KUKA KRL program: EPS_2_251806_MH12A_A_20260223023041.src

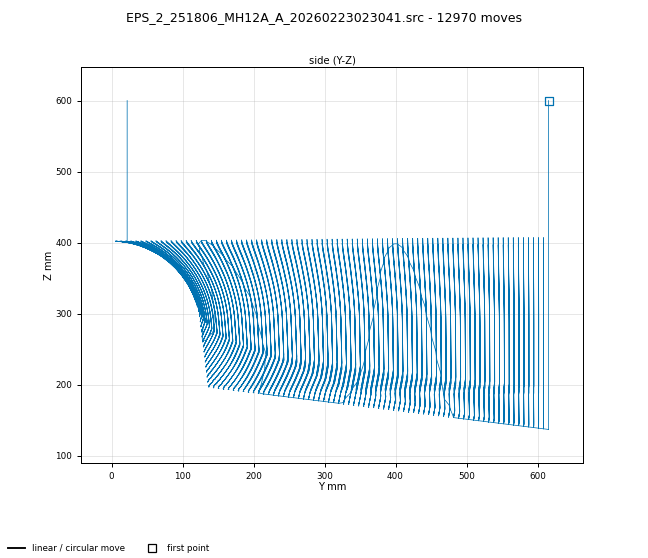
[picture p0: tool path of EPS_2_251806_MH12A_A_20260223023041.src, 12970 of 12972 moves have a stored position in this frame; points joined in program order, loops and branches not executed]
&ACCESS RVP
&REL 4
&COMMENT QRS 19112012
&PARAM EDITMASK = *
DEF PART()
EXT BAS (BAS_COMMAND :IN,REAL :IN )
INT I
BAS (#INITMOV,0 )

;KUKA QRS Post kuka4.cps  Date:22-06-2017 !

File_ID=3069

QRS_PRE_INIT()

;Init var - Until changes are made in qrs_pre_init
Outlet_Square_prg=0
Inlet_1_Square_prg=0
Inlet_2_Square_prg=0
Inlet_3_Square_prg=0
Inlet_4_Square_prg=0
Inlet_5_Square_prg=0

Outlet_1={X 0.000, Y 546.330, Z 306.500, B 0.000, E1 0.000 }
Inlet_1={X 0.000, Y 547.040, Z 296.500, B 0.000, E1 180.000 }
Outlet_1_type=201
Inlet_1_type=201
;QRS#1=Sidecore dimensions
;QRS#2=200-8" PVC SDR 35
;QRS#3=200-8" PVC SDR 35
;QRS#4=
;QRS#5=
;QRS#6=
;QRS#7=
;QRS#8=
;QRS#9=12-08 PSX
;QRS#10=12-08 PSX
;QRS#11=
;QRS#12=
;QRS#13=
;QRS#14=
;QRS#15=
;QRS#16=1220x127x686 2,25'
;QRS#17=EPS Height
;QRS#18=407
;QRS#19=*
;QRS#20= UPDATED VERSION 22-06-2017
;QRS#21=*
Outlet_Square=0100
Inlet_1_Square=0100
Inlet_2_Square=0
Inlet_3_Square=0
Inlet_4_Square=0
Inlet_5_Square=0
Mill_Square=1
Outlet_Square_Prg=204
Inlet_1_Square_prg=204

QRS_INIT()

$ADVANCE=5

; T1
PTP {E1 173.588,E2 173.588}
PTP {X 0,Y 615.517,A -85,B 0,C 180,E1 173.588,E2 173.588,E3 0,E4 0,E5 0,E6 0}
QRS_SPEED_INIT()
LIN {X 0,Y 615.517,Z 600,A -85,B 0,C 180,E1 173.588,E2 173.588,E3 0,E4 0,E5 0,E6 0} C_VEL
LIN {X 0,Y 615.517,Z 146.874,A -85,B 0,C 180,E1 173.588,E2 173.588} C_VEL
LIN {X 0,Y 615.517,Z 138.695,A -85,B 0,C 180,E1 173.588,E2 173.588} C_VEL
LIN {X 0,Y 615.495,Z 136.695,A -85,B 0,C 180,E1 173.402,E2 173.402} C_VEL
LIN {X 0,Y 615.467,Z 136.688,A -85,B 0,C 180,E1 170.801,E2 170.801} C_VEL
LIN {X 0,Y 615.466,Z 136.688,A -85,B 0,C 180,E1 168.806,E2 168.806} C_VEL
LIN {X 0,Y 615.457,Z 136.695,A -85,B 0,C 180,E1 166.125,E2 166.125} C_VEL
LIN {X 0,Y 615.494,Z 136.691,A -85,B 0,C 180,E1 163.413,E2 163.413} C_VEL
LIN {X 0,Y 615.453,Z 136.69,A -85,B 0,C 180,E1 160.661,E2 160.661} C_VEL
LIN {X 0,Y 615.451,Z 136.691,A -85,B 0,C 180,E1 158.567,E2 158.567} C_VEL
LIN {X 0,Y 615.477,Z 136.698,A -85,B 0,C 180,E1 155.99,E2 155.99} C_VEL
LIN {X 0,Y 615.465,Z 136.688,A -85,B 0,C 180,E1 152.956,E2 152.956} C_VEL
LIN {X 0,Y 615.449,Z 136.693,A -85,B 0,C 180,E1 150.592,E2 150.592} C_VEL
LIN {X 0,Y 615.494,Z 136.693,A -85,B 0,C 180,E1 147.666,E2 147.666} C_VEL
LIN {X 0,Y 615.473,Z 136.687,A -85,B 0,C 180,E1 145.184,E2 145.184} C_VEL
LIN {X 0,Y 615.452,Z 136.691,A -85,B 0,C 180,E1 142.755,E2 142.755} C_VEL
LIN {X 0,Y 615.496,Z 136.698,A -85,B 0,C 180,E1 139.908,E2 139.908} C_VEL
LIN {X 0,Y 615.494,Z 136.689,A -85,B 0,C 180,E1 137.647,E2 137.647} C_VEL
LIN {X 0,Y 615.455,Z 136.69,A -85,B 0,C 180,E1 134.928,E2 134.928} C_VEL
LIN {X 0,Y 615.496,Z 136.701,A -85,B 0,C 180,E1 132.081,E2 132.081} C_VEL
LIN {X 0,Y 615.494,Z 136.689,A -85,B 0,C 180,E1 129.748,E2 129.748} C_VEL
LIN {X 0,Y 615.466,Z 136.687,A -85,B 0,C 180,E1 127.242,E2 127.242} C_VEL
LIN {X 0,Y 615.458,Z 136.694,A -85,B 0,C 180,E1 124.696,E2 124.696} C_VEL
LIN {X 0,Y 615.487,Z 136.699,A -85,B 0,C 180,E1 122.33,E2 122.33} C_VEL
LIN {X 0,Y 615.472,Z 136.686,A -85,B 0,C 180,E1 119.406,E2 119.406} C_VEL
LIN {X 0,Y 615.455,Z 136.691,A -85,B 0,C 180,E1 117.038,E2 117.038} C_VEL
LIN {X 0,Y 615.454,Z 136.692,A -85,B 0,C 180,E1 114.992,E2 114.992} C_VEL
LIN {X 0,Y 615.491,Z 136.694,A -85,B 0,C 180,E1 112.135,E2 112.135} C_VEL
LIN {X 0,Y 615.491,Z 136.885,A -85,B 0,C 180,E1 110.293,E2 110.293} C_VEL
LIN {X 0,Y 615.493,Z 154.026,A -85,B 0,C 180,E1 107.612,E2 107.612} C_VEL
LIN {X 0,Y 615.449,Z 171.874,A -85,B 0,C 180,E1 104.888,E2 104.888} C_VEL
LIN {X 0,Y 615.436,Z 185.406,A -85,B 0,C 180,E1 102.866,E2 102.866} C_VEL
LIN {X 0,Y 615.435,Z 186.907,A -85,B 0,C 180,E1 102.803,E2 102.803} C_VEL
LIN {X 0,Y 615.497,Z 292.675,A -85,B 0,C 180,E1 101.547,E2 101.547} C_VEL
LIN {X 0,Y 615.498,Z 305.242,A -85,B 0,C 180,E1 101.276,E2 101.276} C_VEL
LIN {X 0,Y 615.497,Z 318.527,A -85,B 0,C 180,E1 100.845,E2 100.845} C_VEL
LIN {X 0,Y 615.491,Z 329.577,A -85,B 0,C 180,E1 100.36,E2 100.36} C_VEL
LIN {X 0,Y 615.492,Z 341.312,A -85,B 0,C 180,E1 99.696,E2 99.696} C_VEL
LIN {X 0,Y 615.499,Z 351.774,A -85,B 0,C 180,E1 98.95,E2 98.95} C_VEL
LIN {X 0,Y 615.498,Z 360.336,A -85,B 0,C 180,E1 98.205,E2 98.205} C_VEL
LIN {X 0,Y 615.497,Z 368.213,A -85,B 0,C 180,E1 97.38,E2 97.38} C_VEL
LIN {X 0,Y 615.497,Z 375.902,A -85,B 0,C 180,E1 96.392,E2 96.392} C_VEL
LIN {X 0,Y 615.497,Z 382.96,A -85,B 0,C 180,E1 95.241,E2 95.241} C_VEL
LIN {X 0,Y 615.494,Z 387.659,A -85,B 0,C 180,E1 94.256,E2 94.256} C_VEL
LIN {X 0,Y 615.494,Z 391.256,A -85,B 0,C 180,E1 93.273,E2 93.273} C_VEL
LIN {X 0,Y 615.496,Z 393.116,A -85,B 0,C 180,E1 92.617,E2 92.617} C_VEL
LIN {X 0,Y 615.499,Z 394.533,A -85,B 0,C 180,E1 91.963,E2 91.963} C_VEL
LIN {X 0,Y 615.496,Z 396.142,A -85,B 0,C 180,E1 90.654,E2 90.654} C_VEL
LIN {X 0,Y 615.495,Z 396.384,A -85,B 0,C 180,E1 90,E2 90} C_VEL
LIN {X 0,Y 615.495,Z 396.205,A -85,B 0,C 180,E1 89.345,E2 89.345} C_VEL
LIN {X 0,Y 615.499,Z 394.682,A -85,B 0,C 180,E1 88.037,E2 88.037} C_VEL
LIN {X 0,Y 615.498,Z 393.341,A -85,B 0,C 180,E1 87.382,E2 87.382} C_VEL
LIN {X 0,Y 615.496,Z 390.493,A -85,B 0,C 180,E1 86.399,E2 86.399} C_VEL
LIN {X 0,Y 615.498,Z 386.633,A -85,B 0,C 180,E1 85.415,E2 85.415} C_VEL
LIN {X 0,Y 615.498,Z 381.651,A -85,B 0,C 180,E1 84.43,E2 84.43} C_VEL
LIN {X 0,Y 615.496,Z 375.208,A -85,B 0,C 180,E1 83.418,E2 83.418} C_VEL
LIN {X 0,Y 615.497,Z 367.536,A -85,B 0,C 180,E1 82.454,E2 82.454} C_VEL
LIN {X 0,Y 615.498,Z 357.758,A -85,B 0,C 180,E1 81.463,E2 81.463} C_VEL
LIN {X 0,Y 615.498,Z 347.492,A -85,B 0,C 180,E1 80.636,E2 80.636} C_VEL
LIN {X 0,Y 615.486,Z 335.93,A -85,B 0,C 180,E1 79.889,E2 79.889} C_VEL
LIN {X 0,Y 615.497,Z 324.023,A -85,B 0,C 180,E1 79.291,E2 79.291} C_VEL
LIN {X 0,Y 615.498,Z 311.157,A -85,B 0,C 180,E1 78.807,E2 78.807} C_VEL
LIN {X 0,Y 615.497,Z 298.557,A -85,B 0,C 180,E1 78.473,E2 78.473} C_VEL
LIN {X 0,Y 615.495,Z 285.433,A -85,B 0,C 180,E1 78.265,E2 78.265} C_VEL
LIN {X 0,Y 615.429,Z 186.202,A -85,B 0,C 180,E1 77.091,E2 77.091} C_VEL
LIN {X 0,Y 615.434,Z 184.751,A -85,B 0,C 180,E1 76.966,E2 76.966} C_VEL
LIN {X 0,Y 615.496,Z 166.877,A -85,B 0,C 180,E1 74.265,E2 74.265} C_VEL
LIN {X 0,Y 615.455,Z 149.286,A -85,B 0,C 180,E1 71.565,E2 71.565} C_VEL
LIN {X 0,Y 615.497,Z 136.85,A -85,B 0,C 180,E1 69.608,E2 69.608} C_VEL
LIN {X 0,Y 615.464,Z 136.695,A -85,B 0,C 180,E1 67.155,E2 67.155} C_VEL
LIN {X 0,Y 615.483,Z 136.684,A -85,B 0,C 180,E1 64.433,E2 64.433} C_VEL
LIN {X 0,Y 615.489,Z 136.699,A -85,B 0,C 180,E1 61.55,E2 61.55} C_VEL
LIN {X 0,Y 615.46,Z 136.69,A -85,B 0,C 180,E1 58.919,E2 58.919} C_VEL
LIN {X 0,Y 615.488,Z 136.683,A -85,B 0,C 180,E1 56.466,E2 56.466} C_VEL
LIN {X 0,Y 615.481,Z 136.698,A -85,B 0,C 180,E1 53.575,E2 53.575} C_VEL
LIN {X 0,Y 615.458,Z 136.689,A -85,B 0,C 180,E1 50.942,E2 50.942} C_VEL
LIN {X 0,Y 615.489,Z 136.684,A -85,B 0,C 180,E1 48.527,E2 48.527} C_VEL
LIN {X 0,Y 615.497,Z 136.701,A -85,B 0,C 180,E1 45.852,E2 45.852} C_VEL
LIN {X 0,Y 615.46,Z 136.689,A -85,B 0,C 180,E1 43.046,E2 43.046} C_VEL
LIN {X 0,Y 615.489,Z 136.684,A -85,B 0,C 180,E1 40.607,E2 40.607} C_VEL
LIN {X 0,Y 615.484,Z 136.702,A -85,B 0,C 180,E1 38.013,E2 38.013} C_VEL
LIN {X 0,Y 615.465,Z 136.696,A -85,B 0,C 180,E1 35.618,E2 35.618} C_VEL
LIN {X 0,Y 615.456,Z 136.69,A -85,B 0,C 180,E1 33.238,E2 33.238} C_VEL
LIN {X 0,Y 615.473,Z 136.686,A -85,B 0,C 180,E1 30.921,E2 30.921} C_VEL
LIN {X 0,Y 615.48,Z 136.698,A -85,B 0,C 180,E1 27.916,E2 27.916} C_VEL
LIN {X 0,Y 615.456,Z 136.693,A -85,B 0,C 180,E1 25.565,E2 25.565} C_VEL
LIN {X 0,Y 615.488,Z 136.684,A -85,B 0,C 180,E1 22.845,E2 22.845} C_VEL
LIN {X 0,Y 615.481,Z 136.698,A -85,B 0,C 180,E1 20.033,E2 20.033} C_VEL
LIN {X 0,Y 615.469,Z 136.697,A -85,B 0,C 180,E1 17.958,E2 17.958} C_VEL
LIN {X 0,Y 615.464,Z 136.696,A -85,B 0,C 180,E1 15.906,E2 15.906} C_VEL
LIN {X 0,Y 615.466,Z 136.687,A -85,B 0,C 180,E1 13.202,E2 13.202} C_VEL
LIN {X 0,Y 615.494,Z 136.694,A -85,B 0,C 180,E1 10.527,E2 10.527} C_VEL
LIN {X 0,Y 615.457,Z 136.695,A -85,B 0,C 180,E1 7.876,E2 7.876} C_VEL
LIN {X 0,Y 615.469,Z 136.687,A -85,B 0,C 180,E1 5.241,E2 5.241} C_VEL
LIN {X 0,Y 615.494,Z 136.695,A -85,B 0,C 180,E1 2.618,E2 2.618} C_VEL
LIN {X 0,Y 615.457,Z 136.695,A -85,B 0,C 180,E1 0,E2 0} C_VEL
LIN {X 0,Y 615.464,Z 136.688,A -85,B 0,C 180,E1 -2.618,E2 -2.618} C_VEL
LIN {X 0,Y 615.494,Z 136.693,A -85,B 0,C 180,E1 -5.241,E2 -5.241} C_VEL
LIN {X 0,Y 615.456,Z 136.696,A -85,B 0,C 180,E1 -7.876,E2 -7.876} C_VEL
LIN {X 0,Y 615.463,Z 136.688,A -85,B 0,C 180,E1 -10.527,E2 -10.527} C_VEL
LIN {X 0,Y 615.495,Z 136.695,A -85,B 0,C 180,E1 -13.201,E2 -13.201} C_VEL
LIN {X 0,Y 615.451,Z 136.694,A -85,B 0,C 180,E1 -15.906,E2 -15.906} C_VEL
LIN {X 0,Y 615.448,Z 136.694,A -85,B 0,C 180,E1 -17.958,E2 -17.958} C_VEL
LIN {X 0,Y 615.49,Z 136.687,A -85,B 0,C 180,E1 -20.731,E2 -20.731} C_VEL
LIN {X 0,Y 615.464,Z 136.697,A -85,B 0,C 180,E1 -23.557,E2 -23.557} C_VEL
LIN {X 0,Y 615.451,Z 136.695,A -85,B 0,C 180,E1 -25.717,E2 -25.717} C_VEL
LIN {X 0,Y 615.447,Z 136.693,A -85,B 0,C 180,E1 -27.917,E2 -27.917} C_VEL
LIN {X 0,Y 615.449,Z 136.691,A -85,B 0,C 180,E1 -30.162,E2 -30.162} C_VEL
LIN {X 0,Y 615.478,Z 136.687,A -85,B 0,C 180,E1 -32.458,E2 -32.458} C_VEL
LIN {X 0,Y 615.495,Z 136.692,A -85,B 0,C 180,E1 -34.815,E2 -34.815} C_VEL
LIN {X 0,Y 615.474,Z 136.698,A -85,B 0,C 180,E1 -37.243,E2 -37.243} C_VEL
LIN {X 0,Y 615.445,Z 136.693,A -85,B 0,C 180,E1 -39.754,E2 -39.754} C_VEL
LIN {X 0,Y 615.478,Z 136.688,A -85,B 0,C 180,E1 -42.354,E2 -42.354} C_VEL
LIN {X 0,Y 615.482,Z 136.699,A -85,B 0,C 180,E1 -45.069,E2 -45.069} C_VEL
LIN {X 0,Y 615.444,Z 136.694,A -85,B 0,C 180,E1 -47.644,E2 -47.644} C_VEL
LIN {X 0,Y 615.476,Z 136.688,A -85,B 0,C 180,E1 -50.25,E2 -50.25} C_VEL
LIN {X 0,Y 615.47,Z 136.698,A -85,B 0,C 180,E1 -53.066,E2 -53.066} C_VEL
LIN {X 0,Y 615.45,Z 136.696,A -85,B 0,C 180,E1 -55.305,E2 -55.305} C_VEL
LIN {X 0,Y 615.443,Z 136.693,A -85,B 0,C 180,E1 -57.676,E2 -57.676} C_VEL
LIN {X 0,Y 615.482,Z 136.688,A -85,B 0,C 180,E1 -60.207,E2 -60.207} C_VEL
LIN {X 0,Y 615.467,Z 136.698,A -85,B 0,C 180,E1 -62.959,E2 -62.959} C_VEL
LIN {X 0,Y 615.46,Z 136.697,A -85,B 0,C 180,E1 -65.007,E2 -65.007} C_VEL
LIN {X 0,Y 615.446,Z 136.696,A -85,B 0,C 180,E1 -67.154,E2 -67.154} C_VEL
LIN {X 0,Y 615.494,Z 136.913,A -85,B 0,C 180,E1 -68.7,E2 -68.7} C_VEL
LIN {X 0,Y 615.486,Z 153.668,A -85,B 0,C 180,E1 -71.181,E2 -71.181} C_VEL
LIN {X 0,Y 615.486,Z 173.832,A -85,B 0,C 180,E1 -74.095,E2 -74.095} C_VEL
LIN {X 0,Y 615.479,Z 193.975,A -85,B 0,C 180,E1 -76.967,E2 -76.967} C_VEL
LIN {X 0,Y 615.486,Z 195.337,A -85,B 0,C 180,E1 -77.114,E2 -77.114} C_VEL
LIN {X 0,Y 615.487,Z 202.259,A -85,B 0,C 180,E1 -77.218,E2 -77.218} C_VEL
LIN {X 0,Y 615.498,Z 302.827,A -85,B 0,C 180,E1 -78.411,E2 -78.411} C_VEL
LIN {X 0,Y 615.498,Z 315.341,A -85,B 0,C 180,E1 -78.682,E2 -78.682} C_VEL
LIN {X 0,Y 615.496,Z 328.502,A -85,B 0,C 180,E1 -79.109,E2 -79.109} C_VEL
LIN {X 0,Y 615.489,Z 340.476,A -85,B 0,C 180,E1 -79.639,E2 -79.639} C_VEL
LIN {X 0,Y 615.495,Z 351.993,A -85,B 0,C 180,E1 -80.304,E2 -80.304} C_VEL
LIN {X 0,Y 615.499,Z 362.34,A -85,B 0,C 180,E1 -81.05,E2 -81.05} C_VEL
LIN {X 0,Y 615.497,Z 370.811,A -85,B 0,C 180,E1 -81.794,E2 -81.794} C_VEL
LIN {X 0,Y 615.498,Z 378.605,A -85,B 0,C 180,E1 -82.619,E2 -82.619} C_VEL
LIN {X 0,Y 615.496,Z 386.202,A -85,B 0,C 180,E1 -83.608,E2 -83.608} C_VEL
LIN {X 0,Y 615.498,Z 393.204,A -85,B 0,C 180,E1 -84.759,E2 -84.759} C_VEL
LIN {X 0,Y 615.494,Z 397.85,A -85,B 0,C 180,E1 -85.743,E2 -85.743} C_VEL
LIN {X 0,Y 615.494,Z 401.398,A -85,B 0,C 180,E1 -86.727,E2 -86.727} C_VEL
LIN {X 0,Y 615.497,Z 403.232,A -85,B 0,C 180,E1 -87.382,E2 -87.382} C_VEL
LIN {X 0,Y 615.499,Z 404.607,A -85,B 0,C 180,E1 -88.037,E2 -88.037} C_VEL
LIN {X 0,Y 615.496,Z 406.173,A -85,B 0,C 180,E1 -89.345,E2 -89.345} C_VEL
LIN {X 0,Y 615.494,Z 406.389,A -85,B 0,C 180,E1 -90,E2 -90} C_VEL
LIN {X 0,Y 615.495,Z 405.58,A -85,B 0,C 180,E1 -91.308,E2 -91.308} C_VEL
LIN {X 0,Y 615.499,Z 404.608,A -85,B 0,C 180,E1 -91.963,E2 -91.963} C_VEL
LIN {X 0,Y 615.497,Z 403.234,A -85,B 0,C 180,E1 -92.617,E2 -92.617} C_VEL
LIN {X 0,Y 615.496,Z 400.351,A -85,B 0,C 180,E1 -93.6,E2 -93.6} C_VEL
LIN {X 0,Y 615.498,Z 396.443,A -85,B 0,C 180,E1 -94.584,E2 -94.584} C_VEL
LIN {X 0,Y 615.499,Z 391.407,A -85,B 0,C 180,E1 -95.569,E2 -95.569} C_VEL
LIN {X 0,Y 615.496,Z 384.87,A -85,B 0,C 180,E1 -96.583,E2 -96.583} C_VEL
LIN {X 0,Y 615.497,Z 377.137,A -85,B 0,C 180,E1 -97.545,E2 -97.545} C_VEL
LIN {X 0,Y 615.498,Z 369.05,A -85,B 0,C 180,E1 -98.371,E2 -98.371} C_VEL
LIN {X 0,Y 615.499,Z 359.174,A -85,B 0,C 180,E1 -99.198,E2 -99.198} C_VEL
LIN {X 0,Y 615.492,Z 347.989,A -85,B 0,C 180,E1 -99.945,E2 -99.945} C_VEL
LIN {X 0,Y 615.493,Z 337.033,A -85,B 0,C 180,E1 -100.526,E2 -100.526} C_VEL
LIN {X 0,Y 615.499,Z 324.425,A -85,B 0,C 180,E1 -101.042,E2 -101.042} C_VEL
LIN {X 0,Y 615.499,Z 312.087,A -85,B 0,C 180,E1 -101.401,E2 -101.401} C_VEL
LIN {X 0,Y 615.499,Z 298.504,A -85,B 0,C 180,E1 -101.651,E2 -101.651} C_VEL
LIN {X 0,Y 615.486,Z 195.821,A -85,B 0,C 180,E1 -102.865,E2 -102.865} C_VEL
LIN {X 0,Y 615.484,Z 194.624,A -85,B 0,C 180,E1 -102.949,E2 -102.949} C_VEL
LIN {X 0,Y 615.491,Z 175.021,A -85,B 0,C 180,E1 -105.734,E2 -105.734} C_VEL
LIN {X 0,Y 615.476,Z 155.169,A -85,B 0,C 180,E1 -108.601,E2 -108.601} C_VEL
LIN {X 0,Y 615.494,Z 137.129,A -85,B 0,C 180,E1 -111.255,E2 -111.255} C_VEL
LIN {X 0,Y 615.498,Z 136.727,A -85,B 0,C 180,E1 -111.431,E2 -111.431} C_VEL
LIN {X 0,Y 615.446,Z 136.692,A -85,B 0,C 180,E1 -114.273,E2 -114.273} C_VEL
LIN {X 0,Y 615.441,Z 136.693,A -85,B 0,C 180,E1 -116.445,E2 -116.445} C_VEL
LIN {X 0,Y 615.444,Z 136.695,A -85,B 0,C 180,E1 -118.659,E2 -118.659} C_VEL
LIN {X 0,Y 615.476,Z 136.699,A -85,B 0,C 180,E1 -121.084,E2 -121.084} C_VEL
LIN {X 0,Y 615.456,Z 136.69,A -85,B 0,C 180,E1 -124.023,E2 -124.023} C_VEL
LIN {X 0,Y 615.442,Z 136.694,A -85,B 0,C 180,E1 -126.427,E2 -126.427} C_VEL
LIN {X 0,Y 615.487,Z 136.699,A -85,B 0,C 180,E1 -129.062,E2 -129.062} C_VEL
LIN {X 0,Y 615.495,Z 136.69,A -85,B 0,C 180,E1 -131.472,E2 -131.472} C_VEL
LIN {X 0,Y 615.445,Z 136.692,A -85,B 0,C 180,E1 -134.152,E2 -134.152} C_VEL
LIN {X 0,Y 615.485,Z 136.699,A -85,B 0,C 180,E1 -136.951,E2 -136.951} C_VEL
LIN {X 0,Y 615.494,Z 136.689,A -85,B 0,C 180,E1 -139.394,E2 -139.394} C_VEL
LIN {X 0,Y 615.448,Z 136.691,A -85,B 0,C 180,E1 -141.991,E2 -141.991} C_VEL
LIN {X 0,Y 615.448,Z 136.695,A -85,B 0,C 180,E1 -144.381,E2 -144.381} C_VEL
LIN {X 0,Y 615.47,Z 136.7,A -85,B 0,C 180,E1 -146.763,E2 -146.763} C_VEL
LIN {X 0,Y 615.492,Z 136.695,A -85,B 0,C 180,E1 -149.08,E2 -149.08} C_VEL
LIN {X 0,Y 615.471,Z 136.688,A -85,B 0,C 180,E1 -151.549,E2 -151.549} C_VEL
LIN {X 0,Y 615.466,Z 136.689,A -85,B 0,C 180,E1 -153.555,E2 -153.555} C_VEL
LIN {X 0,Y 615.445,Z 136.692,A -85,B 0,C 180,E1 -155.997,E2 -155.997} C_VEL
LIN {X 0,Y 615.473,Z 136.698,A -85,B 0,C 180,E1 -158.568,E2 -158.568} C_VEL
LIN {X 0,Y 615.475,Z 136.688,A -85,B 0,C 180,E1 -161.394,E2 -161.394} C_VEL
LIN {X 0,Y 615.459,Z 136.689,A -85,B 0,C 180,E1 -163.572,E2 -163.572} C_VEL
LIN {X 0,Y 615.45,Z 136.695,A -85,B 0,C 180,E1 -166.125,E2 -166.125} C_VEL
LIN {X 0,Y 615.493,Z 136.696,A -85,B 0,C 180,E1 -168.807,E2 -168.807} C_VEL
LIN {X 0,Y 615.457,Z 136.69,A -85,B 0,C 180,E1 -171.463,E2 -171.463} C_VEL
LIN {X 0,Y 615.461,Z 136.689,A -85,B 0,C 180,E1 -173.443,E2 -173.443} C_VEL
LIN {X 0,Y 615.454,Z 136.695,A -85,B 0,C 180,E1 -176.071,E2 -176.071} C_VEL
LIN {X 0,Y 615.495,Z 136.695,A -85,B 0,C 180,E1 -178.691,E2 -178.691} C_VEL
LIN {X 0,Y 615.465,Z 136.688,A -85,B 0,C 180,E1 -181.309,E2 -181.309} C_VEL
LIN {X 0,Y 615.453,Z 136.695,A -85,B 0,C 180,E1 -183.929,E2 -183.929} C_VEL
LIN {X 0,Y 615.495,Z 136.695,A -85,B 0,C 180,E1 -186.598,E2 -186.598} C_VEL
LIN {X 0,Y 614.801,Z 136.835,A -85,B 0,C 180,E1 -187.144,E2 -187.144} C_VEL
LIN {X 0,Y 611.954,Z 137.255,A -85,B 0,C 180,E1 -188.03,E2 -188.03} C_VEL
LIN {X 0,Y 609.562,Z 137.562,A -85,B 0,C 180,E1 -188.742,E2 -188.742} C_VEL
LIN {X 0,Y 608.526,Z 137.679,A -85,B 0,C 180,E1 -189.292,E2 -189.292} C_VEL
LIN {X 0,Y 608.437,Z 137.689,A -85,B 0,C 180,E1 -189.478,E2 -189.478} C_VEL
LIN {X 0,Y 608.44,Z 137.693,A -85,B 0,C 180,E1 -192,E2 -192} C_VEL
LIN {X 0,Y 608.472,Z 137.689,A -85,B 0,C 180,E1 -194.721,E2 -194.721} C_VEL
LIN {X 0,Y 608.427,Z 137.691,A -85,B 0,C 180,E1 -197.477,E2 -197.477} C_VEL
LIN {X 0,Y 608.428,Z 137.691,A -85,B 0,C 180,E1 -199.572,E2 -199.572} C_VEL
LIN {X 0,Y 608.447,Z 137.69,A -85,B 0,C 180,E1 -201.692,E2 -201.692} C_VEL
LIN {X 0,Y 608.448,Z 137.692,A -85,B 0,C 180,E1 -204.571,E2 -204.571} C_VEL
LIN {X 0,Y 608.43,Z 137.691,A -85,B 0,C 180,E1 -207.519,E2 -207.519} C_VEL
LIN {X 0,Y 608.476,Z 137.692,A -85,B 0,C 180,E1 -209.976,E2 -209.976} C_VEL
LIN {X 0,Y 608.443,Z 137.689,A -85,B 0,C 180,E1 -212.881,E2 -212.881} C_VEL
LIN {X 0,Y 608.422,Z 137.691,A -85,B 0,C 180,E1 -215.279,E2 -215.279} C_VEL
LIN {X 0,Y 608.465,Z 137.693,A -85,B 0,C 180,E1 -218.242,E2 -218.242} C_VEL
LIN {X 0,Y 608.474,Z 137.69,A -85,B 0,C 180,E1 -220.334,E2 -220.334} C_VEL
LIN {X 0,Y 608.428,Z 137.69,A -85,B 0,C 180,E1 -222.962,E2 -222.962} C_VEL
LIN {X 0,Y 608.455,Z 137.694,A -85,B 0,C 180,E1 -225.737,E2 -225.737} C_VEL
LIN {X 0,Y 608.452,Z 137.688,A -85,B 0,C 180,E1 -228.659,E2 -228.659} C_VEL
LIN {X 0,Y 608.466,Z 137.695,A -85,B 0,C 180,E1 -231.76,E2 -231.76} C_VEL
LIN {X 0,Y 608.437,Z 137.689,A -85,B 0,C 180,E1 -234.723,E2 -234.723} C_VEL
LIN {X 0,Y 608.442,Z 137.69,A -85,B 0,C 180,E1 -237.121,E2 -237.121} C_VEL
LIN {X 0,Y 608.474,Z 137.69,A -85,B 0,C 180,E1 -240.028,E2 -240.028} C_VEL
LIN {X 0,Y 608.456,Z 137.687,A -85,B 0,C 180,E1 -242.797,E2 -242.797} C_VEL
LIN {X 0,Y 608.444,Z 137.695,A -85,B 0,C 180,E1 -245.429,E2 -245.429} C_VEL
LIN {X 0,Y 608.459,Z 137.688,A -85,B 0,C 180,E1 -248.309,E2 -248.309} C_VEL
LIN {X 0,Y 608.495,Z 137.899,A -85,B 0,C 180,E1 -249.629,E2 -249.629} C_VEL
LIN {X 0,Y 608.506,Z 154.095,A -85,B 0,C 180,E1 -252.179,E2 -252.179} C_VEL
LIN {X 0,Y 608.448,Z 171.991,A -85,B 0,C 180,E1 -254.937,E2 -254.937} C_VEL
LIN {X 0,Y 608.455,Z 185.735,A -85,B 0,C 180,E1 -257.005,E2 -257.005} C_VEL
LIN {X 0,Y 608.528,Z 188.555,A -85,B 0,C 180,E1 -257.07,E2 -257.07} C_VEL
LIN {X 0,Y 608.557,Z 292.826,A -85,B 0,C 180,E1 -258.32,E2 -258.32} C_VEL
LIN {X 0,Y 608.538,Z 306.134,A -85,B 0,C 180,E1 -258.615,E2 -258.615} C_VEL
LIN {X 0,Y 608.529,Z 319.355,A -85,B 0,C 180,E1 -259.055,E2 -259.055} C_VEL
LIN {X 0,Y 608.503,Z 331.379,A -85,B 0,C 180,E1 -259.604,E2 -259.604} C_VEL
LIN {X 0,Y 608.506,Z 342.798,A -85,B 0,C 180,E1 -260.276,E2 -260.276} C_VEL
LIN {X 0,Y 608.474,Z 353.09,A -85,B 0,C 180,E1 -261.03,E2 -261.03} C_VEL
LIN {X 0,Y 608.464,Z 362.354,A -85,B 0,C 180,E1 -261.866,E2 -261.866} C_VEL
LIN {X 0,Y 608.466,Z 371.327,A -85,B 0,C 180,E1 -262.868,E2 -262.868} C_VEL
LIN {X 0,Y 608.444,Z 378.558,A -85,B 0,C 180,E1 -263.867,E2 -263.867} C_VEL
LIN {X 0,Y 608.462,Z 383.437,A -85,B 0,C 180,E1 -264.699,E2 -264.699} C_VEL
LIN {X 0,Y 608.439,Z 388.18,A -85,B 0,C 180,E1 -265.695,E2 -265.695} C_VEL
LIN {X 0,Y 608.425,Z 391.813,A -85,B 0,C 180,E1 -266.689,E2 -266.689} C_VEL
LIN {X 0,Y 608.425,Z 393.692,A -85,B 0,C 180,E1 -267.352,E2 -267.352} C_VEL
LIN {X 0,Y 608.444,Z 395.127,A -85,B 0,C 180,E1 -268.015,E2 -268.015} C_VEL
LIN {X 0,Y 608.439,Z 396.752,A -85,B 0,C 180,E1 -269.338,E2 -269.338} C_VEL
LIN {X 0,Y 608.435,Z 396.995,A -85,B 0,C 180,E1 -270,E2 -270} C_VEL
LIN {X 0,Y 608.438,Z 396.815,A -85,B 0,C 180,E1 -270.662,E2 -270.662} C_VEL
LIN {X 0,Y 608.444,Z 395.276,A -85,B 0,C 180,E1 -271.986,E2 -271.986} C_VEL
LIN {X 0,Y 608.426,Z 393.918,A -85,B 0,C 180,E1 -272.648,E2 -272.648} C_VEL
LIN {X 0,Y 608.449,Z 391.041,A -85,B 0,C 180,E1 -273.643,E2 -273.643} C_VEL
LIN {X 0,Y 608.433,Z 387.142,A -85,B 0,C 180,E1 -274.638,E2 -274.638} C_VEL
LIN {X 0,Y 608.45,Z 382.111,A -85,B 0,C 180,E1 -275.635,E2 -275.635} C_VEL
LIN {X 0,Y 608.441,Z 375.794,A -85,B 0,C 180,E1 -276.633,E2 -276.633} C_VEL
LIN {X 0,Y 608.475,Z 367.877,A -85,B 0,C 180,E1 -277.633,E2 -277.633} C_VEL
LIN {X 0,Y 608.472,Z 358.035,A -85,B 0,C 180,E1 -278.636,E2 -278.636} C_VEL
LIN {X 0,Y 608.48,Z 347.713,A -85,B 0,C 180,E1 -279.473,E2 -279.473} C_VEL
LIN {X 0,Y 608.483,Z 336.099,A -85,B 0,C 180,E1 -280.229,E2 -280.229} C_VEL
LIN {X 0,Y 608.529,Z 324.86,A -85,B 0,C 180,E1 -280.803,E2 -280.803} C_VEL
LIN {X 0,Y 608.538,Z 312.26,A -85,B 0,C 180,E1 -281.29,E2 -281.29} C_VEL
LIN {X 0,Y 608.539,Z 299.559,A -85,B 0,C 180,E1 -281.639,E2 -281.639} C_VEL
LIN {X 0,Y 608.564,Z 287.289,A -85,B 0,C 180,E1 -281.85,E2 -281.85} C_VEL
LIN {X 0,Y 608.484,Z 186.214,A -85,B 0,C 180,E1 -283.059,E2 -283.059} C_VEL
LIN {X 0,Y 608.425,Z 184.884,A -85,B 0,C 180,E1 -283.187,E2 -283.187} C_VEL
LIN {X 0,Y 608.487,Z 166.979,A -85,B 0,C 180,E1 -285.921,E2 -285.921} C_VEL
LIN {X 0,Y 608.466,Z 150.674,A -85,B 0,C 180,E1 -288.445,E2 -288.445} C_VEL
LIN {X 0,Y 608.505,Z 137.841,A -85,B 0,C 180,E1 -290.471,E2 -290.471} C_VEL
LIN {X 0,Y 608.438,Z 137.69,A -85,B 0,C 180,E1 -293.124,E2 -293.124} C_VEL
LIN {X 0,Y 608.477,Z 137.686,A -85,B 0,C 180,E1 -295.721,E2 -295.721} C_VEL
LIN {X 0,Y 608.468,Z 137.691,A -85,B 0,C 180,E1 -298.619,E2 -298.619} C_VEL
LIN {X 0,Y 608.442,Z 137.688,A -85,B 0,C 180,E1 -301.317,E2 -301.317} C_VEL
LIN {X 0,Y 608.475,Z 137.687,A -85,B 0,C 180,E1 -303.735,E2 -303.735} C_VEL
LIN {X 0,Y 608.477,Z 137.692,A -85,B 0,C 180,E1 -306.09,E2 -306.09} C_VEL
LIN {X 0,Y 608.427,Z 137.695,A -85,B 0,C 180,E1 -308.59,E2 -308.59} C_VEL
LIN {X 0,Y 608.454,Z 137.687,A -85,B 0,C 180,E1 -311.341,E2 -311.341} C_VEL
LIN {X 0,Y 608.461,Z 137.695,A -85,B 0,C 180,E1 -314.264,E2 -314.264} C_VEL
LIN {X 0,Y 608.431,Z 137.69,A -85,B 0,C 180,E1 -317.038,E2 -317.038} C_VEL
LIN {X 0,Y 608.457,Z 137.691,A -85,B 0,C 180,E1 -319.697,E2 -319.697} C_VEL
LIN {X 0,Y 608.46,Z 137.693,A -85,B 0,C 180,E1 -322.253,E2 -322.253} C_VEL
LIN {X 0,Y 608.427,Z 137.691,A -85,B 0,C 180,E1 -324.721,E2 -324.721} C_VEL
LIN {X 0,Y 608.465,Z 137.688,A -85,B 0,C 180,E1 -327.476,E2 -327.476} C_VEL
LIN {X 0,Y 608.455,Z 137.693,A -85,B 0,C 180,E1 -330.22,E2 -330.22} C_VEL
LIN {X 0,Y 608.458,Z 137.687,A -85,B 0,C 180,E1 -332.794,E2 -332.794} C_VEL
LIN {X 0,Y 608.479,Z 137.695,A -85,B 0,C 180,E1 -335.845,E2 -335.845} C_VEL
LIN {X 0,Y 608.451,Z 137.69,A -85,B 0,C 180,E1 -338.308,E2 -338.308} C_VEL
LIN {X 0,Y 608.448,Z 137.689,A -85,B 0,C 180,E1 -341.13,E2 -341.13} C_VEL
LIN {X 0,Y 608.45,Z 137.695,A -85,B 0,C 180,E1 -343.906,E2 -343.906} C_VEL
LIN {X 0,Y 608.443,Z 137.688,A -85,B 0,C 180,E1 -346.643,E2 -346.643} C_VEL
LIN {X 0,Y 608.469,Z 137.69,A -85,B 0,C 180,E1 -349.35,E2 -349.35} C_VEL
LIN {X 0,Y 608.456,Z 137.691,A -85,B 0,C 180,E1 -352.033,E2 -352.033} C_VEL
LIN {X 0,Y 608.447,Z 137.688,A -85,B 0,C 180,E1 -354.698,E2 -354.698} C_VEL
LIN {X 0,Y 608.482,Z 137.69,A -85,B 0,C 180,E1 -357.352,E2 -357.352} C_VEL
LIN {X 0,Y 608.45,Z 137.691,A -85,B 0,C 180,E1 -360,E2 -360} C_VEL
LIN {X 0,Y 608.458,Z 137.687,A -85,B 0,C 180,E1 -362.648,E2 -362.648} C_VEL
LIN {X 0,Y 608.469,Z 137.693,A -85,B 0,C 180,E1 -365.302,E2 -365.302} C_VEL
LIN {X 0,Y 608.423,Z 137.693,A -85,B 0,C 180,E1 -367.968,E2 -367.968} C_VEL
LIN {X 0,Y 608.429,Z 137.692,A -85,B 0,C 180,E1 -369.978,E2 -369.978} C_VEL
LIN {X 0,Y 608.462,Z 137.687,A -85,B 0,C 180,E1 -372.677,E2 -372.677} C_VEL
LIN {X 0,Y 608.464,Z 137.695,A -85,B 0,C 180,E1 -375.406,E2 -375.406} C_VEL
LIN {X 0,Y 608.449,Z 137.695,A -85,B 0,C 180,E1 -377.477,E2 -377.477} C_VEL
LIN {X 0,Y 608.435,Z 137.689,A -85,B 0,C 180,E1 -380.275,E2 -380.275} C_VEL
LIN {X 0,Y 608.447,Z 137.697,A -85,B 0,C 180,E1 -383.124,E2 -383.124} C_VEL
LIN {X 0,Y 608.444,Z 137.691,A -85,B 0,C 180,E1 -385.718,E2 -385.718} C_VEL
LIN {X 0,Y 608.429,Z 137.69,A -85,B 0,C 180,E1 -388.268,E2 -388.268} C_VEL
LIN {X 0,Y 608.439,Z 137.691,A -85,B 0,C 180,E1 -390.547,E2 -390.547} C_VEL
LIN {X 0,Y 608.448,Z 137.695,A -85,B 0,C 180,E1 -392.88,E2 -392.88} C_VEL
LIN {X 0,Y 608.426,Z 137.697,A -85,B 0,C 180,E1 -395.279,E2 -395.279} C_VEL
LIN {X 0,Y 608.443,Z 137.689,A -85,B 0,C 180,E1 -397.748,E2 -397.748} C_VEL
LIN {X 0,Y 608.437,Z 137.69,A -85,B 0,C 180,E1 -400.329,E2 -400.329} C_VEL
LIN {X 0,Y 608.454,Z 137.692,A -85,B 0,C 180,E1 -403.308,E2 -403.308} C_VEL
LIN {X 0,Y 608.445,Z 137.689,A -85,B 0,C 180,E1 -406.129,E2 -406.129} C_VEL
LIN {X 0,Y 608.456,Z 137.697,A -85,B 0,C 180,E1 -408.824,E2 -408.824} C_VEL
LIN {X 0,Y 608.419,Z 137.693,A -85,B 0,C 180,E1 -411.409,E2 -411.409} C_VEL
LIN {X 0,Y 608.437,Z 137.689,A -85,B 0,C 180,E1 -413.956,E2 -413.956} C_VEL
LIN {X 0,Y 608.465,Z 137.689,A -85,B 0,C 180,E1 -416.33,E2 -416.33} C_VEL
LIN {X 0,Y 608.445,Z 137.699,A -85,B 0,C 180,E1 -418.733,E2 -418.733} C_VEL
LIN {X 0,Y 608.437,Z 137.69,A -85,B 0,C 180,E1 -421.387,E2 -421.387} C_VEL
LIN {X 0,Y 608.433,Z 137.691,A -85,B 0,C 180,E1 -423.964,E2 -423.964} C_VEL
LIN {X 0,Y 608.434,Z 137.697,A -85,B 0,C 180,E1 -426.876,E2 -426.876} C_VEL
LIN {X 0,Y 608.507,Z 137.906,A -85,B 0,C 180,E1 -428.599,E2 -428.599} C_VEL
LIN {X 0,Y 608.525,Z 153.701,A -85,B 0,C 180,E1 -430.958,E2 -430.958} C_VEL
LIN {X 0,Y 608.494,Z 172.794,A -85,B 0,C 180,E1 -433.745,E2 -433.745} C_VEL
LIN {X 0,Y 608.477,Z 191.749,A -85,B 0,C 180,E1 -436.474,E2 -436.474} C_VEL
LIN {X 0,Y 608.497,Z 195.382,A -85,B 0,C 180,E1 -436.963,E2 -436.963} C_VEL
LIN {X 0,Y 608.564,Z 200.51,A -85,B 0,C 180,E1 -437.049,E2 -437.049} C_VEL
LIN {X 0,Y 608.549,Z 302.946,A -85,B 0,C 180,E1 -438.277,E2 -438.277} C_VEL
LIN {X 0,Y 608.547,Z 316.216,A -85,B 0,C 180,E1 -438.572,E2 -438.572} C_VEL
LIN {X 0,Y 608.544,Z 329.332,A -85,B 0,C 180,E1 -439.009,E2 -439.009} C_VEL
LIN {X 0,Y 608.511,Z 340.634,A -85,B 0,C 180,E1 -439.519,E2 -439.519} C_VEL
LIN {X 0,Y 608.486,Z 352.197,A -85,B 0,C 180,E1 -440.191,E2 -440.191} C_VEL
LIN {X 0,Y 608.485,Z 362.593,A -85,B 0,C 180,E1 -440.946,E2 -440.946} C_VEL
LIN {X 0,Y 608.475,Z 371.111,A -85,B 0,C 180,E1 -441.699,E2 -441.699} C_VEL
LIN {X 0,Y 608.471,Z 378.959,A -85,B 0,C 180,E1 -442.534,E2 -442.534} C_VEL
LIN {X 0,Y 608.461,Z 386.286,A -85,B 0,C 180,E1 -443.484,E2 -443.484} C_VEL
LIN {X 0,Y 608.45,Z 391.865,A -85,B 0,C 180,E1 -444.365,E2 -444.365} C_VEL
LIN {X 0,Y 608.432,Z 396.949,A -85,B 0,C 180,E1 -445.362,E2 -445.362} C_VEL
LIN {X 0,Y 608.449,Z 400.895,A -85,B 0,C 180,E1 -446.357,E2 -446.357} C_VEL
LIN {X 0,Y 608.425,Z 403.809,A -85,B 0,C 180,E1 -447.352,E2 -447.352} C_VEL
LIN {X 0,Y 608.444,Z 405.201,A -85,B 0,C 180,E1 -448.014,E2 -448.014} C_VEL
LIN {X 0,Y 608.438,Z 406.783,A -85,B 0,C 180,E1 -449.338,E2 -449.338} C_VEL
LIN {X 0,Y 608.434,Z 407,A -85,B 0,C 180,E1 -450,E2 -450} C_VEL
LIN {X 0,Y 608.448,Z 406.184,A -85,B 0,C 180,E1 -451.323,E2 -451.323} C_VEL
LIN {X 0,Y 608.444,Z 405.202,A -85,B 0,C 180,E1 -451.985,E2 -451.985} C_VEL
LIN {X 0,Y 608.425,Z 403.81,A -85,B 0,C 180,E1 -452.648,E2 -452.648} C_VEL
LIN {X 0,Y 608.449,Z 400.897,A -85,B 0,C 180,E1 -453.642,E2 -453.642} C_VEL
LIN {X 0,Y 608.432,Z 396.952,A -85,B 0,C 180,E1 -454.637,E2 -454.637} C_VEL
LIN {X 0,Y 608.437,Z 390.879,A -85,B 0,C 180,E1 -455.8,E2 -455.8} C_VEL
LIN {X 0,Y 608.462,Z 384.238,A -85,B 0,C 180,E1 -456.799,E2 -456.799} C_VEL
LIN {X 0,Y 608.455,Z 375.993,A -85,B 0,C 180,E1 -457.8,E2 -457.8} C_VEL
LIN {X 0,Y 608.472,Z 367.542,A -85,B 0,C 180,E1 -458.635,E2 -458.635} C_VEL
LIN {X 0,Y 608.479,Z 357.098,A -85,B 0,C 180,E1 -459.473,E2 -459.473} C_VEL
LIN {X 0,Y 608.497,Z 346.765,A -85,B 0,C 180,E1 -460.144,E2 -460.144} C_VEL
LIN {X 0,Y 608.522,Z 335.249,A -85,B 0,C 180,E1 -460.741,E2 -460.741} C_VEL
LIN {X 0,Y 608.533,Z 323.887,A -85,B 0,C 180,E1 -461.192,E2 -461.192} C_VEL
LIN {X 0,Y 608.562,Z 310.377,A -85,B 0,C 180,E1 -461.575,E2 -461.575} C_VEL
LIN {X 0,Y 608.553,Z 297.128,A -85,B 0,C 180,E1 -461.807,E2 -461.807} C_VEL
LIN {X 0,Y 608.547,Z 195.835,A -85,B 0,C 180,E1 -463.014,E2 -463.014} C_VEL
LIN {X 0,Y 608.459,Z 194.758,A -85,B 0,C 180,E1 -463.101,E2 -463.101} C_VEL
LIN {X 0,Y 608.492,Z 175.107,A -85,B 0,C 180,E1 -465.92,E2 -465.92} C_VEL
LIN {X 0,Y 608.493,Z 157.427,A -85,B 0,C 180,E1 -468.496,E2 -468.496} C_VEL
LIN {X 0,Y 608.57,Z 139.436,A -85,B 0,C 180,E1 -471.154,E2 -471.154} C_VEL
LIN {X 0,Y 608.497,Z 137.825,A -85,B 0,C 180,E1 -471.423,E2 -471.423} C_VEL
LIN {X 0,Y 608.432,Z 137.69,A -85,B 0,C 180,E1 -474.142,E2 -474.142} C_VEL
LIN {X 0,Y 608.433,Z 137.691,A -85,B 0,C 180,E1 -476.035,E2 -476.035} C_VEL
LIN {X 0,Y 608.436,Z 137.69,A -85,B 0,C 180,E1 -478.613,E2 -478.613} C_VEL
LIN {X 0,Y 608.457,Z 137.697,A -85,B 0,C 180,E1 -481.316,E2 -481.316} C_VEL
LIN {X 0,Y 608.469,Z 137.688,A -85,B 0,C 180,E1 -483.734,E2 -483.734} C_VEL
LIN {X 0,Y 608.432,Z 137.69,A -85,B 0,C 180,E1 -486.092,E2 -486.092} C_VEL
LIN {X 0,Y 608.418,Z 137.693,A -85,B 0,C 180,E1 -488.59,E2 -488.59} C_VEL
LIN {X 0,Y 608.465,Z 137.693,A -85,B 0,C 180,E1 -491.342,E2 -491.342} C_VEL
LIN {X 0,Y 608.444,Z 137.689,A -85,B 0,C 180,E1 -493.87,E2 -493.87} C_VEL
LIN {X 0,Y 608.453,Z 137.692,A -85,B 0,C 180,E1 -496.691,E2 -496.691} C_VEL
LIN {X 0,Y 608.443,Z 137.69,A -85,B 0,C 180,E1 -499.696,E2 -499.696} C_VEL
LIN {X 0,Y 608.441,Z 137.689,A -85,B 0,C 180,E1 -502.252,E2 -502.252} C_VEL
LIN {X 0,Y 608.481,Z 137.692,A -85,B 0,C 180,E1 -505.088,E2 -505.088} C_VEL
LIN {X 0,Y 608.441,Z 137.689,A -85,B 0,C 180,E1 -507.904,E2 -507.904} C_VEL
LIN {X 0,Y 608.43,Z 137.691,A -85,B 0,C 180,E1 -510.218,E2 -510.218} C_VEL
LIN {X 0,Y 608.477,Z 137.694,A -85,B 0,C 180,E1 -512.79,E2 -512.79} C_VEL
LIN {X 0,Y 608.445,Z 137.688,A -85,B 0,C 180,E1 -515.851,E2 -515.851} C_VEL
LIN {X 0,Y 608.446,Z 137.691,A -85,B 0,C 180,E1 -518.308,E2 -518.308} C_VEL
LIN {X 0,Y 608.46,Z 137.689,A -85,B 0,C 180,E1 -521.282,E2 -521.282} C_VEL
LIN {X 0,Y 608.428,Z 137.691,A -85,B 0,C 180,E1 -523.905,E2 -523.905} C_VEL
LIN {X 0,Y 608.462,Z 137.696,A -85,B 0,C 180,E1 -526.644,E2 -526.644} C_VEL
LIN {X 0,Y 608.449,Z 137.689,A -85,B 0,C 180,E1 -529.35,E2 -529.35} C_VEL
LIN {X 0,Y 608.447,Z 137.69,A -85,B 0,C 180,E1 -532.033,E2 -532.033} C_VEL
LIN {X 0,Y 608.469,Z 137.694,A -85,B 0,C 180,E1 -534.698,E2 -534.698} C_VEL
LIN {X 0,Y 608.456,Z 137.687,A -85,B 0,C 180,E1 -537.352,E2 -537.352} C_VEL
LIN {X 0,Y 608.446,Z 137.691,A -85,B 0,C 180,E1 -540,E2 -540} C_VEL
LIN {X 0,Y 608.483,Z 137.691,A -85,B 0,C 180,E1 -542.648,E2 -542.648} C_VEL
LIN {X 0,Y 608.446,Z 137.688,A -85,B 0,C 180,E1 -545.302,E2 -545.302} C_VEL
LIN {X 0,Y 608.452,Z 137.691,A -85,B 0,C 180,E1 -547.967,E2 -547.967} C_VEL
LIN {X 0,Y 608.437,Z 137.689,A -85,B 0,C 180,E1 -549.478,E2 -549.478} C_VEL
LIN {X 0,Y 607.756,Z 137.78,A -85,B 0,C 180,E1 -550.031,E2 -550.031} C_VEL
LIN {X 0,Y 604.9,Z 138.136,A -85,B 0,C 180,E1 -550.928,E2 -550.928} C_VEL
LIN {X 0,Y 602.5,Z 138.436,A -85,B 0,C 180,E1 -551.65,E2 -551.65} C_VEL
LIN {X 0,Y 601.476,Z 138.564,A -85,B 0,C 180,E1 -552.206,E2 -552.206} C_VEL
LIN {X 0,Y 601.396,Z 138.57,A -85,B 0,C 180,E1 -552.395,E2 -552.395} C_VEL
LIN {X 0,Y 601.42,Z 138.565,A -85,B 0,C 180,E1 -554.897,E2 -554.897} C_VEL
LIN {X 0,Y 601.419,Z 138.564,A -85,B 0,C 180,E1 -556.986,E2 -556.986} C_VEL
LIN {X 0,Y 601.39,Z 138.57,A -85,B 0,C 180,E1 -559.81,E2 -559.81} C_VEL
LIN {X 0,Y 601.447,Z 138.564,A -85,B 0,C 180,E1 -562.617,E2 -562.617} C_VEL
LIN {X 0,Y 601.388,Z 138.568,A -85,B 0,C 180,E1 -564.879,E2 -564.879} C_VEL
LIN {X 0,Y 601.411,Z 138.57,A -85,B 0,C 180,E1 -567.868,E2 -567.868} C_VEL
LIN {X 0,Y 601.44,Z 138.571,A -85,B 0,C 180,E1 -570.164,E2 -570.164} C_VEL
LIN {X 0,Y 601.417,Z 138.565,A -85,B 0,C 180,E1 -572.717,E2 -572.717} C_VEL
LIN {X 0,Y 601.381,Z 138.567,A -85,B 0,C 180,E1 -575.112,E2 -575.112} C_VEL
LIN {X 0,Y 601.422,Z 138.564,A -85,B 0,C 180,E1 -577.42,E2 -577.42} C_VEL
LIN {X 0,Y 601.398,Z 138.577,A -85,B 0,C 180,E1 -579.996,E2 -579.996} C_VEL
LIN {X 0,Y 601.402,Z 138.566,A -85,B 0,C 180,E1 -582.671,E2 -582.671} C_VEL
LIN {X 0,Y 601.391,Z 138.57,A -85,B 0,C 180,E1 -585.48,E2 -585.48} C_VEL
LIN {X 0,Y 601.42,Z 138.566,A -85,B 0,C 180,E1 -588.408,E2 -588.408} C_VEL
LIN {X 0,Y 601.393,Z 138.566,A -85,B 0,C 180,E1 -590.874,E2 -590.874} C_VEL
LIN {X 0,Y 601.394,Z 138.57,A -85,B 0,C 180,E1 -593.418,E2 -593.418} C_VEL
LIN {X 0,Y 601.431,Z 138.568,A -85,B 0,C 180,E1 -596.065,E2 -596.065} C_VEL
LIN {X 0,Y 601.415,Z 138.564,A -85,B 0,C 180,E1 -598.547,E2 -598.547} C_VEL
LIN {X 0,Y 601.418,Z 138.568,A -85,B 0,C 180,E1 -601.374,E2 -601.374} C_VEL
LIN {X 0,Y 601.418,Z 138.568,A -85,B 0,C 180,E1 -604.132,E2 -604.132} C_VEL
LIN {X 0,Y 601.392,Z 138.567,A -85,B 0,C 180,E1 -606.589,E2 -606.589} C_VEL
LIN {X 0,Y 601.433,Z 138.659,A -85,B 0,C 180,E1 -609.479,E2 -609.479} C_VEL
LIN {X 0,Y 601.561,Z 144.033,A -85,B 0,C 180,E1 -610.374,E2 -610.374} C_VEL
LIN {X 0,Y 601.469,Z 162.312,A -85,B 0,C 180,E1 -613.251,E2 -613.251} C_VEL
LIN {X 0,Y 601.432,Z 179.419,A -85,B 0,C 180,E1 -615.906,E2 -615.906} C_VEL
LIN {X 0,Y 601.426,Z 185.736,A -85,B 0,C 180,E1 -616.85,E2 -616.85} C_VEL
LIN {X 0,Y 601.608,Z 188.6,A -85,B 0,C 180,E1 -616.919,E2 -616.919} C_VEL
LIN {X 0,Y 601.629,Z 292.855,A -85,B 0,C 180,E1 -618.183,E2 -618.183} C_VEL
LIN {X 0,Y 601.602,Z 306.153,A -85,B 0,C 180,E1 -618.482,E2 -618.482} C_VEL
LIN {X 0,Y 601.566,Z 319.227,A -85,B 0,C 180,E1 -618.921,E2 -618.921} C_VEL
LIN {X 0,Y 601.511,Z 331.389,A -85,B 0,C 180,E1 -619.482,E2 -619.482} C_VEL
LIN {X 0,Y 601.475,Z 342.808,A -85,B 0,C 180,E1 -620.161,E2 -620.161} C_VEL
LIN {X 0,Y 601.438,Z 353.099,A -85,B 0,C 180,E1 -620.924,E2 -620.924} C_VEL
LIN {X 0,Y 601.411,Z 362.359,A -85,B 0,C 180,E1 -621.77,E2 -621.77} C_VEL
LIN {X 0,Y 601.388,Z 371.332,A -85,B 0,C 180,E1 -622.783,E2 -622.783} C_VEL
LIN {X 0,Y 601.376,Z 378.47,A -85,B 0,C 180,E1 -623.781,E2 -623.781} C_VEL
LIN {X 0,Y 601.372,Z 383.44,A -85,B 0,C 180,E1 -624.636,E2 -624.636} C_VEL
LIN {X 0,Y 601.353,Z 388.182,A -85,B 0,C 180,E1 -625.644,E2 -625.644} C_VEL
LIN {X 0,Y 601.344,Z 391.816,A -85,B 0,C 180,E1 -626.65,E2 -626.65} C_VEL
LIN {X 0,Y 601.324,Z 393.694,A -85,B 0,C 180,E1 -627.321,E2 -627.321} C_VEL
LIN {X 0,Y 601.343,Z 395.127,A -85,B 0,C 180,E1 -627.991,E2 -627.991} C_VEL
LIN {X 0,Y 601.339,Z 396.753,A -85,B 0,C 180,E1 -629.331,E2 -629.331} C_VEL
LIN {X 0,Y 601.336,Z 396.996,A -85,B 0,C 180,E1 -630,E2 -630} C_VEL
LIN {X 0,Y 601.339,Z 396.815,A -85,B 0,C 180,E1 -630.67,E2 -630.67} C_VEL
LIN {X 0,Y 601.343,Z 395.275,A -85,B 0,C 180,E1 -632.01,E2 -632.01} C_VEL
LIN {X 0,Y 601.326,Z 393.916,A -85,B 0,C 180,E1 -632.68,E2 -632.68} C_VEL
LIN {X 0,Y 601.368,Z 391.039,A -85,B 0,C 180,E1 -633.686,E2 -633.686} C_VEL
LIN {X 0,Y 601.337,Z 387.14,A -85,B 0,C 180,E1 -634.693,E2 -634.693} C_VEL
LIN {X 0,Y 601.373,Z 382.109,A -85,B 0,C 180,E1 -635.701,E2 -635.701} C_VEL
LIN {X 0,Y 601.382,Z 375.79,A -85,B 0,C 180,E1 -636.711,E2 -636.711} C_VEL
LIN {X 0,Y 601.396,Z 367.873,A -85,B 0,C 180,E1 -637.723,E2 -637.723} C_VEL
LIN {X 0,Y 601.437,Z 358.029,A -85,B 0,C 180,E1 -638.738,E2 -638.738} C_VEL
LIN {X 0,Y 601.45,Z 347.708,A -85,B 0,C 180,E1 -639.585,E2 -639.585} C_VEL
LIN {X 0,Y 601.49,Z 336.087,A -85,B 0,C 180,E1 -640.349,E2 -640.349} C_VEL
LIN {X 0,Y 601.551,Z 324.849,A -85,B 0,C 180,E1 -640.93,E2 -640.93} C_VEL
LIN {X 0,Y 601.565,Z 312.428,A -85,B 0,C 180,E1 -641.417,E2 -641.417} C_VEL
LIN {X 0,Y 601.607,Z 299.536,A -85,B 0,C 180,E1 -641.775,E2 -641.775} C_VEL
LIN {X 0,Y 601.634,Z 287.25,A -85,B 0,C 180,E1 -641.988,E2 -641.988} C_VEL
LIN {X 0,Y 601.487,Z 186.574,A -85,B 0,C 180,E1 -643.202,E2 -643.202} C_VEL
LIN {X 0,Y 601.392,Z 185.533,A -85,B 0,C 180,E1 -643.258,E2 -643.258} C_VEL
LIN {X 0,Y 601.476,Z 168.095,A -85,B 0,C 180,E1 -645.937,E2 -645.937} C_VEL
LIN {X 0,Y 601.494,Z 150.99,A -85,B 0,C 180,E1 -648.616,E2 -648.616} C_VEL
LIN {X 0,Y 601.483,Z 138.776,A -85,B 0,C 180,E1 -650.568,E2 -650.568} C_VEL
LIN {X 0,Y 601.393,Z 138.567,A -85,B 0,C 180,E1 -653.411,E2 -653.411} C_VEL
LIN {X 0,Y 601.42,Z 138.566,A -85,B 0,C 180,E1 -655.868,E2 -655.868} C_VEL
LIN {X 0,Y 601.426,Z 138.569,A -85,B 0,C 180,E1 -658.627,E2 -658.627} C_VEL
LIN {X 0,Y 601.418,Z 138.563,A -85,B 0,C 180,E1 -661.454,E2 -661.454} C_VEL
LIN {X 0,Y 601.425,Z 138.571,A -85,B 0,C 180,E1 -664.118,E2 -664.118} C_VEL
LIN {X 0,Y 601.399,Z 138.571,A -85,B 0,C 180,E1 -666.583,E2 -666.583} C_VEL
LIN {X 0,Y 601.396,Z 138.566,A -85,B 0,C 180,E1 -669.127,E2 -669.127} C_VEL
LIN {X 0,Y 601.426,Z 138.566,A -85,B 0,C 180,E1 -671.764,E2 -671.764} C_VEL
LIN {X 0,Y 601.422,Z 138.567,A -85,B 0,C 180,E1 -674.535,E2 -674.535} C_VEL
LIN {X 0,Y 601.409,Z 138.565,A -85,B 0,C 180,E1 -677.409,E2 -677.409} C_VEL
LIN {X 0,Y 601.401,Z 138.575,A -85,B 0,C 180,E1 -680.004,E2 -680.004} C_VEL
LIN {X 0,Y 601.426,Z 138.564,A -85,B 0,C 180,E1 -682.618,E2 -682.618} C_VEL
LIN {X 0,Y 601.4,Z 138.564,A -85,B 0,C 180,E1 -685.067,E2 -685.067} C_VEL
LIN {X 0,Y 601.433,Z 138.564,A -85,B 0,C 180,E1 -687.484,E2 -687.484} C_VEL
LIN {X 0,Y 601.422,Z 138.572,A -85,B 0,C 180,E1 -689.851,E2 -689.851} C_VEL
LIN {X 0,Y 601.414,Z 138.57,A -85,B 0,C 180,E1 -692.132,E2 -692.132} C_VEL
LIN {X 0,Y 601.391,Z 138.568,A -85,B 0,C 180,E1 -695.121,E2 -695.121} C_VEL
LIN {X 0,Y 601.411,Z 138.568,A -85,B 0,C 180,E1 -697.393,E2 -697.393} C_VEL
LIN {X 0,Y 601.394,Z 138.571,A -85,B 0,C 180,E1 -700.19,E2 -700.19} C_VEL
LIN {X 0,Y 601.422,Z 138.564,A -85,B 0,C 180,E1 -703.014,E2 -703.014} C_VEL
LIN {X 0,Y 601.413,Z 138.572,A -85,B 0,C 180,E1 -705.908,E2 -705.908} C_VEL
LIN {X 0,Y 601.41,Z 138.565,A -85,B 0,C 180,E1 -708.541,E2 -708.541} C_VEL
LIN {X 0,Y 601.434,Z 138.565,A -85,B 0,C 180,E1 -711.262,E2 -711.262} C_VEL
LIN {X 0,Y 601.391,Z 138.572,A -85,B 0,C 180,E1 -713.963,E2 -713.963} C_VEL
LIN {X 0,Y 601.412,Z 138.564,A -85,B 0,C 180,E1 -716.65,E2 -716.65} C_VEL
LIN {X 0,Y 601.455,Z 138.566,A -85,B 0,C 180,E1 -719.33,E2 -719.33} C_VEL
LIN {X 0,Y 601.4,Z 138.569,A -85,B 0,C 180,E1 -722.009,E2 -722.009} C_VEL
LIN {X 0,Y 601.403,Z 138.565,A -85,B 0,C 180,E1 -724.692,E2 -724.692} C_VEL
LIN {X 0,Y 601.444,Z 138.57,A -85,B 0,C 180,E1 -727.385,E2 -727.385} C_VEL
LIN {X 0,Y 601.41,Z 138.565,A -85,B 0,C 180,E1 -730.095,E2 -730.095} C_VEL
LIN {X 0,Y 601.41,Z 138.567,A -85,B 0,C 180,E1 -732.828,E2 -732.828} C_VEL
LIN {X 0,Y 601.401,Z 138.571,A -85,B 0,C 180,E1 -735.592,E2 -735.592} C_VEL
LIN {X 0,Y 601.386,Z 138.571,A -85,B 0,C 180,E1 -737.689,E2 -737.689} C_VEL
LIN {X 0,Y 601.415,Z 138.565,A -85,B 0,C 180,E1 -740.522,E2 -740.522} C_VEL
LIN {X 0,Y 601.406,Z 138.572,A -85,B 0,C 180,E1 -743.411,E2 -743.411} C_VEL
LIN {X 0,Y 601.388,Z 138.568,A -85,B 0,C 180,E1 -746.365,E2 -746.365} C_VEL
LIN {X 0,Y 601.431,Z 138.566,A -85,B 0,C 180,E1 -748.79,E2 -748.79} C_VEL
LIN {X 0,Y 601.387,Z 138.569,A -85,B 0,C 180,E1 -751.728,E2 -751.728} C_VEL
LIN {X 0,Y 601.414,Z 138.564,A -85,B 0,C 180,E1 -754.119,E2 -754.119} C_VEL
LIN {X 0,Y 601.429,Z 138.566,A -85,B 0,C 180,E1 -757.383,E2 -757.383} C_VEL
LIN {X 0,Y 601.393,Z 138.567,A -85,B 0,C 180,E1 -759.997,E2 -759.997} C_VEL
LIN {X 0,Y 601.407,Z 138.57,A -85,B 0,C 180,E1 -762.671,E2 -762.671} C_VEL
LIN {X 0,Y 601.395,Z 138.569,A -85,B 0,C 180,E1 -765.48,E2 -765.48} C_VEL
LIN {X 0,Y 601.418,Z 138.567,A -85,B 0,C 180,E1 -768.408,E2 -768.408} C_VEL
LIN {X 0,Y 601.424,Z 138.573,A -85,B 0,C 180,E1 -770.875,E2 -770.875} C_VEL
LIN {X 0,Y 601.391,Z 138.569,A -85,B 0,C 180,E1 -773.417,E2 -773.417} C_VEL
LIN {X 0,Y 601.427,Z 138.563,A -85,B 0,C 180,E1 -776.066,E2 -776.066} C_VEL
LIN {X 0,Y 601.395,Z 138.572,A -85,B 0,C 180,E1 -779.057,E2 -779.057} C_VEL
LIN {X 0,Y 601.397,Z 138.567,A -85,B 0,C 180,E1 -781.372,E2 -781.372} C_VEL
LIN {X 0,Y 601.412,Z 138.567,A -85,B 0,C 180,E1 -784.133,E2 -784.133} C_VEL
LIN {X 0,Y 601.387,Z 138.577,A -85,B 0,C 180,E1 -786.589,E2 -786.589} C_VEL
LIN {X 0,Y 601.454,Z 138.791,A -85,B 0,C 180,E1 -788.471,E2 -788.471} C_VEL
LIN {X 0,Y 601.589,Z 148.944,A -85,B 0,C 180,E1 -790.019,E2 -790.019} C_VEL
LIN {X 0,Y 601.505,Z 169.158,A -85,B 0,C 180,E1 -793.016,E2 -793.016} C_VEL
LIN {X 0,Y 601.468,Z 189.7,A -85,B 0,C 180,E1 -796.016,E2 -796.016} C_VEL
LIN {X 0,Y 601.46,Z 195.373,A -85,B 0,C 180,E1 -796.808,E2 -796.808} C_VEL
LIN {X 0,Y 601.669,Z 198.721,A -85,B 0,C 180,E1 -796.877,E2 -796.877} C_VEL
LIN {X 0,Y 601.622,Z 302.946,A -85,B 0,C 180,E1 -798.14,E2 -798.14} C_VEL
LIN {X 0,Y 601.591,Z 316.217,A -85,B 0,C 180,E1 -798.438,E2 -798.438} C_VEL
LIN {X 0,Y 601.549,Z 327.923,A -85,B 0,C 180,E1 -798.826,E2 -798.826} C_VEL
LIN {X 0,Y 601.53,Z 338.924,A -85,B 0,C 180,E1 -799.311,E2 -799.311} C_VEL
LIN {X 0,Y 601.481,Z 349.58,A -85,B 0,C 180,E1 -799.906,E2 -799.906} C_VEL
LIN {X 0,Y 601.448,Z 360.475,A -85,B 0,C 180,E1 -800.669,E2 -800.669} C_VEL
LIN {X 0,Y 601.429,Z 371.111,A -85,B 0,C 180,E1 -801.601,E2 -801.601} C_VEL
LIN {X 0,Y 601.418,Z 378.959,A -85,B 0,C 180,E1 -802.446,E2 -802.446} C_VEL
LIN {X 0,Y 601.37,Z 386.224,A -85,B 0,C 180,E1 -803.398,E2 -803.398} C_VEL
LIN {X 0,Y 601.372,Z 391.865,A -85,B 0,C 180,E1 -804.299,E2 -804.299} C_VEL
LIN {X 0,Y 601.336,Z 396.949,A -85,B 0,C 180,E1 -805.307,E2 -805.307} C_VEL
LIN {X 0,Y 601.368,Z 400.895,A -85,B 0,C 180,E1 -806.314,E2 -806.314} C_VEL
LIN {X 0,Y 601.325,Z 403.808,A -85,B 0,C 180,E1 -807.32,E2 -807.32} C_VEL
LIN {X 0,Y 601.343,Z 405.201,A -85,B 0,C 180,E1 -807.99,E2 -807.99} C_VEL
LIN {X 0,Y 601.339,Z 406.784,A -85,B 0,C 180,E1 -809.33,E2 -809.33} C_VEL
LIN {X 0,Y 601.335,Z 407,A -85,B 0,C 180,E1 -810,E2 -810} C_VEL
LIN {X 0,Y 601.347,Z 406.185,A -85,B 0,C 180,E1 -811.339,E2 -811.339} C_VEL
LIN {X 0,Y 601.343,Z 405.203,A -85,B 0,C 180,E1 -812.009,E2 -812.009} C_VEL
LIN {X 0,Y 601.325,Z 403.81,A -85,B 0,C 180,E1 -812.679,E2 -812.679} C_VEL
LIN {X 0,Y 601.368,Z 400.897,A -85,B 0,C 180,E1 -813.685,E2 -813.685} C_VEL
LIN {X 0,Y 601.336,Z 396.951,A -85,B 0,C 180,E1 -814.692,E2 -814.692} C_VEL
LIN {X 0,Y 601.372,Z 390.88,A -85,B 0,C 180,E1 -815.869,E2 -815.869} C_VEL
LIN {X 0,Y 601.381,Z 384.239,A -85,B 0,C 180,E1 -816.879,E2 -816.879} C_VEL
LIN {X 0,Y 601.4,Z 375.994,A -85,B 0,C 180,E1 -817.892,E2 -817.892} C_VEL
LIN {X 0,Y 601.436,Z 367.543,A -85,B 0,C 180,E1 -818.737,E2 -818.737} C_VEL
LIN {X 0,Y 601.449,Z 357.1,A -85,B 0,C 180,E1 -819.585,E2 -819.585} C_VEL
LIN {X 0,Y 601.476,Z 346.767,A -85,B 0,C 180,E1 -820.264,E2 -820.264} C_VEL
LIN {X 0,Y 601.538,Z 335.903,A -85,B 0,C 180,E1 -820.836,E2 -820.836} C_VEL
LIN {X 0,Y 601.565,Z 323.388,A -85,B 0,C 180,E1 -821.34,E2 -821.34} C_VEL
LIN {X 0,Y 601.607,Z 310.376,A -85,B 0,C 180,E1 -821.71,E2 -821.71} C_VEL
LIN {X 0,Y 601.623,Z 297.128,A -85,B 0,C 180,E1 -821.945,E2 -821.945} C_VEL
LIN {X 0,Y 601.574,Z 196.277,A -85,B 0,C 180,E1 -823.157,E2 -823.157} C_VEL
LIN {X 0,Y 601.453,Z 195.108,A -85,B 0,C 180,E1 -823.213,E2 -823.213} C_VEL
LIN {X 0,Y 601.481,Z 176.296,A -85,B 0,C 180,E1 -825.937,E2 -825.937} C_VEL
LIN {X 0,Y 601.52,Z 159.65,A -85,B 0,C 180,E1 -828.388,E2 -828.388} C_VEL
LIN {X 0,Y 601.635,Z 140.625,A -85,B 0,C 180,E1 -831.23,E2 -831.23} C_VEL
LIN {X 0,Y 601.423,Z 138.638,A -85,B 0,C 180,E1 -831.597,E2 -831.597} C_VEL
LIN {X 0,Y 601.397,Z 138.566,A -85,B 0,C 180,E1 -834.284,E2 -834.284} C_VEL
LIN {X 0,Y 601.385,Z 138.568,A -85,B 0,C 180,E1 -836.364,E2 -836.364} C_VEL
LIN {X 0,Y 601.403,Z 138.568,A -85,B 0,C 180,E1 -838.782,E2 -838.782} C_VEL
LIN {X 0,Y 601.394,Z 138.57,A -85,B 0,C 180,E1 -841.726,E2 -841.726} C_VEL
LIN {X 0,Y 601.414,Z 138.564,A -85,B 0,C 180,E1 -844.118,E2 -844.118} C_VEL
LIN {X 0,Y 601.389,Z 138.569,A -85,B 0,C 180,E1 -846.583,E2 -846.583} C_VEL
LIN {X 0,Y 601.431,Z 138.566,A -85,B 0,C 180,E1 -849.534,E2 -849.534} C_VEL
LIN {X 0,Y 601.407,Z 138.566,A -85,B 0,C 180,E1 -851.765,E2 -851.765} C_VEL
LIN {X 0,Y 601.389,Z 138.569,A -85,B 0,C 180,E1 -854.532,E2 -854.532} C_VEL
LIN {X 0,Y 601.405,Z 138.57,A -85,B 0,C 180,E1 -857.408,E2 -857.408} C_VEL
LIN {X 0,Y 601.389,Z 138.567,A -85,B 0,C 180,E1 -860.003,E2 -860.003} C_VEL
LIN {X 0,Y 601.425,Z 138.566,A -85,B 0,C 180,E1 -862.617,E2 -862.617} C_VEL
LIN {X 0,Y 601.435,Z 138.57,A -85,B 0,C 180,E1 -865.069,E2 -865.069} C_VEL
LIN {X 0,Y 601.421,Z 138.565,A -85,B 0,C 180,E1 -867.484,E2 -867.484} C_VEL
LIN {X 0,Y 601.39,Z 138.567,A -85,B 0,C 180,E1 -869.855,E2 -869.855} C_VEL
LIN {X 0,Y 601.385,Z 138.568,A -85,B 0,C 180,E1 -872.131,E2 -872.131} C_VEL
LIN {X 0,Y 601.407,Z 138.568,A -85,B 0,C 180,E1 -874.381,E2 -874.381} C_VEL
LIN {X 0,Y 601.404,Z 138.572,A -85,B 0,C 180,E1 -876.589,E2 -876.589} C_VEL
LIN {X 0,Y 601.415,Z 138.565,A -85,B 0,C 180,E1 -879.478,E2 -879.478} C_VEL
LIN {X 0,Y 601.382,Z 138.571,A -85,B 0,C 180,E1 -882.311,E2 -882.311} C_VEL
LIN {X 0,Y 601.418,Z 138.568,A -85,B 0,C 180,E1 -885.103,E2 -885.103} C_VEL
LIN {X 0,Y 601.393,Z 138.567,A -85,B 0,C 180,E1 -887.857,E2 -887.857} C_VEL
LIN {X 0,Y 601.407,Z 138.565,A -85,B 0,C 180,E1 -889.905,E2 -889.905} C_VEL
LIN {X 0,Y 601.444,Z 138.571,A -85,B 0,C 180,E1 -892.615,E2 -892.615} C_VEL
LIN {X 0,Y 601.404,Z 138.565,A -85,B 0,C 180,E1 -895.308,E2 -895.308} C_VEL
LIN {X 0,Y 601.396,Z 138.569,A -85,B 0,C 180,E1 -897.991,E2 -897.991} C_VEL
LIN {X 0,Y 601.453,Z 138.567,A -85,B 0,C 180,E1 -900.67,E2 -900.67} C_VEL
LIN {X 0,Y 601.41,Z 138.564,A -85,B 0,C 180,E1 -903.35,E2 -903.35} C_VEL
LIN {X 0,Y 601.387,Z 138.571,A -85,B 0,C 180,E1 -906.037,E2 -906.037} C_VEL
LIN {X 0,Y 601.432,Z 138.566,A -85,B 0,C 180,E1 -908.738,E2 -908.738} C_VEL
LIN {X 0,Y 601.416,Z 138.564,A -85,B 0,C 180,E1 -911.459,E2 -911.459} C_VEL
LIN {X 0,Y 601.396,Z 138.57,A -85,B 0,C 180,E1 -912.395,E2 -912.395} C_VEL
LIN {X 0,Y 600.738,Z 138.651,A -85,B 0,C 180,E1 -912.954,E2 -912.954} C_VEL
LIN {X 0,Y 597.888,Z 139.006,A -85,B 0,C 180,E1 -913.862,E2 -913.862} C_VEL
LIN {X 0,Y 595.474,Z 139.309,A -85,B 0,C 180,E1 -914.592,E2 -914.592} C_VEL
LIN {X 0,Y 594.433,Z 139.434,A -85,B 0,C 180,E1 -915.156,E2 -915.156} C_VEL
LIN {X 0,Y 594.346,Z 139.444,A -85,B 0,C 180,E1 -915.347,E2 -915.347} C_VEL
LIN {X 0,Y 594.375,Z 139.441,A -85,B 0,C 180,E1 -917.194,E2 -917.194} C_VEL
LIN {X 0,Y 594.365,Z 139.449,A -85,B 0,C 180,E1 -920.054,E2 -920.054} C_VEL
LIN {X 0,Y 594.363,Z 139.443,A -85,B 0,C 180,E1 -922.967,E2 -922.967} C_VEL
LIN {X 0,Y 594.351,Z 139.444,A -85,B 0,C 180,E1 -925.194,E2 -925.194} C_VEL
LIN {X 0,Y 594.374,Z 139.442,A -85,B 0,C 180,E1 -927.528,E2 -927.528} C_VEL
LIN {X 0,Y 594.389,Z 139.446,A -85,B 0,C 180,E1 -930.331,E2 -930.331} C_VEL
LIN {X 0,Y 594.368,Z 139.441,A -85,B 0,C 180,E1 -932.951,E2 -932.951} C_VEL
LIN {X 0,Y 594.344,Z 139.444,A -85,B 0,C 180,E1 -935.41,E2 -935.41} C_VEL
LIN {X 0,Y 594.38,Z 139.449,A -85,B 0,C 180,E1 -937.941,E2 -937.941} C_VEL
LIN {X 0,Y 594.37,Z 139.442,A -85,B 0,C 180,E1 -940.823,E2 -940.823} C_VEL
LIN {X 0,Y 594.358,Z 139.443,A -85,B 0,C 180,E1 -943.301,E2 -943.301} C_VEL
LIN {X 0,Y 594.355,Z 139.45,A -85,B 0,C 180,E1 -946.162,E2 -946.162} C_VEL
LIN {X 0,Y 594.376,Z 139.442,A -85,B 0,C 180,E1 -948.537,E2 -948.537} C_VEL
LIN {X 0,Y 594.367,Z 139.443,A -85,B 0,C 180,E1 -951.298,E2 -951.298} C_VEL
LIN {X 0,Y 594.366,Z 139.452,A -85,B 0,C 180,E1 -953.758,E2 -953.758} C_VEL
LIN {X 0,Y 594.376,Z 139.444,A -85,B 0,C 180,E1 -956.24,E2 -956.24} C_VEL
LIN {X 0,Y 594.364,Z 139.442,A -85,B 0,C 180,E1 -958.651,E2 -958.651} C_VEL
LIN {X 0,Y 594.376,Z 139.442,A -85,B 0,C 180,E1 -961.044,E2 -961.044} C_VEL
LIN {X 0,Y 594.39,Z 139.446,A -85,B 0,C 180,E1 -963.977,E2 -963.977} C_VEL
LIN {X 0,Y 594.377,Z 139.443,A -85,B 0,C 180,E1 -966.296,E2 -966.296} C_VEL
LIN {X 0,Y 594.403,Z 139.524,A -85,B 0,C 180,E1 -969.361,E2 -969.361} C_VEL
LIN {X 0,Y 594.619,Z 142.918,A -85,B 0,C 180,E1 -969.956,E2 -969.956} C_VEL
LIN {X 0,Y 594.488,Z 160.813,A -85,B 0,C 180,E1 -972.81,E2 -972.81} C_VEL
LIN {X 0,Y 594.403,Z 176.472,A -85,B 0,C 180,E1 -975.274,E2 -975.274} C_VEL
LIN {X 0,Y 594.402,Z 185.737,A -85,B 0,C 180,E1 -976.692,E2 -976.692} C_VEL
LIN {X 0,Y 594.706,Z 188.645,A -85,B 0,C 180,E1 -976.764,E2 -976.764} C_VEL
LIN {X 0,Y 594.689,Z 292.884,A -85,B 0,C 180,E1 -978.043,E2 -978.043} C_VEL
LIN {X 0,Y 594.635,Z 306.172,A -85,B 0,C 180,E1 -978.345,E2 -978.345} C_VEL
LIN {X 0,Y 594.594,Z 318.162,A -85,B 0,C 180,E1 -978.748,E2 -978.748} C_VEL
LIN {X 0,Y 594.543,Z 329.775,A -85,B 0,C 180,E1 -979.271,E2 -979.271} C_VEL
LIN {X 0,Y 594.483,Z 341.538,A -85,B 0,C 180,E1 -979.958,E2 -979.958} C_VEL
LIN {X 0,Y 594.414,Z 352.048,A -85,B 0,C 180,E1 -980.73,E2 -980.73} C_VEL
LIN {X 0,Y 594.384,Z 360.651,A -85,B 0,C 180,E1 -981.501,E2 -981.501} C_VEL
LIN {X 0,Y 594.347,Z 368.577,A -85,B 0,C 180,E1 -982.356,E2 -982.356} C_VEL
LIN {X 0,Y 594.305,Z 376.396,A -85,B 0,C 180,E1 -983.39,E2 -983.39} C_VEL
LIN {X 0,Y 594.289,Z 383.443,A -85,B 0,C 180,E1 -984.572,E2 -984.572} C_VEL
LIN {X 0,Y 594.27,Z 388.185,A -85,B 0,C 180,E1 -985.592,E2 -985.592} C_VEL
LIN {X 0,Y 594.267,Z 391.818,A -85,B 0,C 180,E1 -986.61,E2 -986.61} C_VEL
LIN {X 0,Y 594.225,Z 393.696,A -85,B 0,C 180,E1 -987.289,E2 -987.289} C_VEL
LIN {X 0,Y 594.242,Z 395.127,A -85,B 0,C 180,E1 -987.967,E2 -987.967} C_VEL
LIN {X 0,Y 594.24,Z 396.754,A -85,B 0,C 180,E1 -989.323,E2 -989.323} C_VEL
LIN {X 0,Y 594.236,Z 396.996,A -85,B 0,C 180,E1 -990,E2 -990} C_VEL
LIN {X 0,Y 594.239,Z 396.815,A -85,B 0,C 180,E1 -990.678,E2 -990.678} C_VEL
LIN {X 0,Y 594.242,Z 395.275,A -85,B 0,C 180,E1 -992.034,E2 -992.034} C_VEL
LIN {X 0,Y 594.226,Z 393.914,A -85,B 0,C 180,E1 -992.712,E2 -992.712} C_VEL
LIN {X 0,Y 594.289,Z 391.037,A -85,B 0,C 180,E1 -993.729,E2 -993.729} C_VEL
LIN {X 0,Y 594.241,Z 387.138,A -85,B 0,C 180,E1 -994.749,E2 -994.749} C_VEL
LIN {X 0,Y 594.3,Z 382.106,A -85,B 0,C 180,E1 -995.769,E2 -995.769} C_VEL
LIN {X 0,Y 594.316,Z 375.786,A -85,B 0,C 180,E1 -996.791,E2 -996.791} C_VEL
LIN {X 0,Y 594.346,Z 367.869,A -85,B 0,C 180,E1 -997.816,E2 -997.816} C_VEL
LIN {X 0,Y 594.381,Z 358.022,A -85,B 0,C 180,E1 -998.842,E2 -998.842} C_VEL
LIN {X 0,Y 594.434,Z 347.703,A -85,B 0,C 180,E1 -999.699,E2 -999.699} C_VEL
LIN {X 0,Y 594.499,Z 336.076,A -85,B 0,C 180,E1 -1000.472,E2 -1000.472} C_VEL
LIN {X 0,Y 594.546,Z 324.207,A -85,B 0,C 180,E1 -1001.088,E2 -1001.088} C_VEL
LIN {X 0,Y 594.612,Z 311.231,A -85,B 0,C 180,E1 -1001.591,E2 -1001.591} C_VEL
LIN {X 0,Y 594.667,Z 298.597,A -85,B 0,C 180,E1 -1001.936,E2 -1001.936} C_VEL
LIN {X 0,Y 594.701,Z 285.451,A -85,B 0,C 180,E1 -1002.152,E2 -1002.152} C_VEL
LIN {X 0,Y 594.545,Z 187.154,A -85,B 0,C 180,E1 -1003.349,E2 -1003.349} C_VEL
LIN {X 0,Y 594.381,Z 185.527,A -85,B 0,C 180,E1 -1003.418,E2 -1003.418} C_VEL
LIN {X 0,Y 594.47,Z 166.972,A -85,B 0,C 180,E1 -1006.307,E2 -1006.307} C_VEL
LIN {X 0,Y 594.595,Z 147.949,A -85,B 0,C 180,E1 -1009.327,E2 -1009.327} C_VEL
LIN {X 0,Y 594.427,Z 139.623,A -85,B 0,C 180,E1 -1010.684,E2 -1010.684} C_VEL
LIN {X 0,Y 594.377,Z 139.442,A -85,B 0,C 180,E1 -1013.704,E2 -1013.704} C_VEL
LIN {X 0,Y 594.379,Z 139.446,A -85,B 0,C 180,E1 -1016.699,E2 -1016.699} C_VEL
LIN {X 0,Y 594.377,Z 139.442,A -85,B 0,C 180,E1 -1018.998,E2 -1018.998} C_VEL
LIN {X 0,Y 594.378,Z 139.441,A -85,B 0,C 180,E1 -1021.642,E2 -1021.642} C_VEL
LIN {X 0,Y 594.371,Z 139.446,A -85,B 0,C 180,E1 -1024.58,E2 -1024.58} C_VEL
LIN {X 0,Y 594.379,Z 139.441,A -85,B 0,C 180,E1 -1027.087,E2 -1027.087} C_VEL
LIN {X 0,Y 594.355,Z 139.446,A -85,B 0,C 180,E1 -1029.771,E2 -1029.771} C_VEL
LIN {X 0,Y 594.364,Z 139.449,A -85,B 0,C 180,E1 -1032.375,E2 -1032.375} C_VEL
LIN {X 0,Y 594.361,Z 139.442,A -85,B 0,C 180,E1 -1035.191,E2 -1035.191} C_VEL
LIN {X 0,Y 594.378,Z 139.45,A -85,B 0,C 180,E1 -1038.151,E2 -1038.151} C_VEL
LIN {X 0,Y 594.366,Z 139.448,A -85,B 0,C 180,E1 -1040.319,E2 -1040.319} C_VEL
LIN {X 0,Y 594.377,Z 139.44,A -85,B 0,C 180,E1 -1042.912,E2 -1042.912} C_VEL
LIN {X 0,Y 594.379,Z 139.446,A -85,B 0,C 180,E1 -1045.86,E2 -1045.86} C_VEL
LIN {X 0,Y 594.361,Z 139.444,A -85,B 0,C 180,E1 -1048.649,E2 -1048.649} C_VEL
LIN {X 0,Y 594.378,Z 139.441,A -85,B 0,C 180,E1 -1051.041,E2 -1051.041} C_VEL
LIN {X 0,Y 594.373,Z 139.45,A -85,B 0,C 180,E1 -1053.978,E2 -1053.978} C_VEL
LIN {X 0,Y 594.372,Z 139.444,A -85,B 0,C 180,E1 -1056.295,E2 -1056.295} C_VEL
LIN {X 0,Y 594.404,Z 139.439,A -85,B 0,C 180,E1 -1059.224,E2 -1059.224} C_VEL
LIN {X 0,Y 594.341,Z 139.45,A -85,B 0,C 180,E1 -1062.094,E2 -1062.094} C_VEL
LIN {X 0,Y 594.353,Z 139.446,A -85,B 0,C 180,E1 -1064.219,E2 -1064.219} C_VEL
LIN {X 0,Y 594.368,Z 139.443,A -85,B 0,C 180,E1 -1066.321,E2 -1066.321} C_VEL
LIN {X 0,Y 594.377,Z 139.442,A -85,B 0,C 180,E1 -1069.095,E2 -1069.095} C_VEL
LIN {X 0,Y 594.403,Z 139.444,A -85,B 0,C 180,E1 -1071.843,E2 -1071.843} C_VEL
LIN {X 0,Y 594.375,Z 139.441,A -85,B 0,C 180,E1 -1074.572,E2 -1074.572} C_VEL
LIN {X 0,Y 594.409,Z 139.442,A -85,B 0,C 180,E1 -1077.289,E2 -1077.289} C_VEL
LIN {X 0,Y 594.39,Z 139.442,A -85,B 0,C 180,E1 -1080,E2 -1080} C_VEL
LIN {X 0,Y 594.393,Z 139.439,A -85,B 0,C 180,E1 -1082.711,E2 -1082.711} C_VEL
LIN {X 0,Y 594.389,Z 139.448,A -85,B 0,C 180,E1 -1085.428,E2 -1085.428} C_VEL
LIN {X 0,Y 594.349,Z 139.445,A -85,B 0,C 180,E1 -1088.158,E2 -1088.158} C_VEL
LIN {X 0,Y 594.382,Z 139.445,A -85,B 0,C 180,E1 -1091.075,E2 -1091.075} C_VEL
LIN {X 0,Y 594.364,Z 139.447,A -85,B 0,C 180,E1 -1093.679,E2 -1093.679} C_VEL
LIN {X 0,Y 594.38,Z 139.442,A -85,B 0,C 180,E1 -1096.718,E2 -1096.718} C_VEL
LIN {X 0,Y 594.357,Z 139.453,A -85,B 0,C 180,E1 -1099.335,E2 -1099.335} C_VEL
LIN {X 0,Y 594.352,Z 139.45,A -85,B 0,C 180,E1 -1101.504,E2 -1101.504} C_VEL
LIN {X 0,Y 594.38,Z 139.44,A -85,B 0,C 180,E1 -1104.447,E2 -1104.447} C_VEL
LIN {X 0,Y 594.379,Z 139.445,A -85,B 0,C 180,E1 -1107.527,E2 -1107.527} C_VEL
LIN {X 0,Y 594.36,Z 139.443,A -85,B 0,C 180,E1 -1110.325,E2 -1110.325} C_VEL
LIN {X 0,Y 594.37,Z 139.45,A -85,B 0,C 180,E1 -1112.951,E2 -1112.951} C_VEL
LIN {X 0,Y 594.343,Z 139.448,A -85,B 0,C 180,E1 -1115.41,E2 -1115.41} C_VEL
LIN {X 0,Y 594.37,Z 139.441,A -85,B 0,C 180,E1 -1117.942,E2 -1117.942} C_VEL
LIN {X 0,Y 594.369,Z 139.449,A -85,B 0,C 180,E1 -1120.822,E2 -1120.822} C_VEL
LIN {X 0,Y 594.347,Z 139.449,A -85,B 0,C 180,E1 -1123.301,E2 -1123.301} C_VEL
LIN {X 0,Y 594.356,Z 139.444,A -85,B 0,C 180,E1 -1126.162,E2 -1126.162} C_VEL
LIN {X 0,Y 594.371,Z 139.447,A -85,B 0,C 180,E1 -1129.179,E2 -1129.179} C_VEL
LIN {X 0,Y 594.37,Z 139.441,A -85,B 0,C 180,E1 -1132.059,E2 -1132.059} C_VEL
LIN {X 0,Y 594.347,Z 139.453,A -85,B 0,C 180,E1 -1134.677,E2 -1134.677} C_VEL
LIN {X 0,Y 594.371,Z 139.447,A -85,B 0,C 180,E1 -1137.09,E2 -1137.09} C_VEL
LIN {X 0,Y 594.365,Z 139.442,A -85,B 0,C 180,E1 -1139.676,E2 -1139.676} C_VEL
LIN {X 0,Y 594.376,Z 139.449,A -85,B 0,C 180,E1 -1142.54,E2 -1142.54} C_VEL
LIN {X 0,Y 594.37,Z 139.449,A -85,B 0,C 180,E1 -1144.807,E2 -1144.807} C_VEL
LIN {X 0,Y 594.346,Z 139.447,A -85,B 0,C 180,E1 -1147.766,E2 -1147.766} C_VEL
LIN {X 0,Y 594.396,Z 139.592,A -85,B 0,C 180,E1 -1148.316,E2 -1148.316} C_VEL
LIN {X 0,Y 594.678,Z 143.898,A -85,B 0,C 180,E1 -1149.009,E2 -1149.009} C_VEL
LIN {X 0,Y 594.551,Z 163.213,A -85,B 0,C 180,E1 -1151.923,E2 -1151.923} C_VEL
LIN {X 0,Y 594.457,Z 182.237,A -85,B 0,C 180,E1 -1154.749,E2 -1154.749} C_VEL
LIN {X 0,Y 594.43,Z 195.364,A -85,B 0,C 180,E1 -1156.649,E2 -1156.649} C_VEL
LIN {X 0,Y 594.768,Z 198.721,A -85,B 0,C 180,E1 -1156.722,E2 -1156.722} C_VEL
LIN {X 0,Y 594.691,Z 302.946,A -85,B 0,C 180,E1 -1157.999,E2 -1157.999} C_VEL
LIN {X 0,Y 594.639,Z 316.218,A -85,B 0,C 180,E1 -1158.301,E2 -1158.301} C_VEL
LIN {X 0,Y 594.587,Z 329.367,A -85,B 0,C 180,E1 -1158.749,E2 -1158.749} C_VEL
LIN {X 0,Y 594.537,Z 340.631,A -85,B 0,C 180,E1 -1159.27,E2 -1159.27} C_VEL
LIN {X 0,Y 594.482,Z 352.2,A -85,B 0,C 180,E1 -1159.958,E2 -1159.958} C_VEL
LIN {X 0,Y 594.414,Z 362.596,A -85,B 0,C 180,E1 -1160.73,E2 -1160.73} C_VEL
LIN {X 0,Y 594.383,Z 371.111,A -85,B 0,C 180,E1 -1161.5,E2 -1161.5} C_VEL
LIN {X 0,Y 594.347,Z 378.959,A -85,B 0,C 180,E1 -1162.355,E2 -1162.355} C_VEL
LIN {X 0,Y 594.283,Z 386.813,A -85,B 0,C 180,E1 -1163.408,E2 -1163.408} C_VEL
LIN {X 0,Y 594.289,Z 393.679,A -85,B 0,C 180,E1 -1164.571,E2 -1164.571} C_VEL
LIN {X 0,Y 594.27,Z 398.371,A -85,B 0,C 180,E1 -1165.591,E2 -1165.591} C_VEL
LIN {X 0,Y 594.267,Z 401.956,A -85,B 0,C 180,E1 -1166.61,E2 -1166.61} C_VEL
LIN {X 0,Y 594.226,Z 403.808,A -85,B 0,C 180,E1 -1167.288,E2 -1167.288} C_VEL
LIN {X 0,Y 594.242,Z 405.2,A -85,B 0,C 180,E1 -1167.966,E2 -1167.966} C_VEL
LIN {X 0,Y 594.239,Z 406.784,A -85,B 0,C 180,E1 -1169.322,E2 -1169.322} C_VEL
LIN {X 0,Y 594.236,Z 407,A -85,B 0,C 180,E1 -1170,E2 -1170} C_VEL
LIN {X 0,Y 594.247,Z 406.185,A -85,B 0,C 180,E1 -1171.355,E2 -1171.355} C_VEL
LIN {X 0,Y 594.242,Z 405.202,A -85,B 0,C 180,E1 -1172.033,E2 -1172.033} C_VEL
LIN {X 0,Y 594.226,Z 403.81,A -85,B 0,C 180,E1 -1172.711,E2 -1172.711} C_VEL
LIN {X 0,Y 594.289,Z 400.897,A -85,B 0,C 180,E1 -1173.729,E2 -1173.729} C_VEL
LIN {X 0,Y 594.241,Z 396.951,A -85,B 0,C 180,E1 -1174.748,E2 -1174.748} C_VEL
LIN {X 0,Y 594.304,Z 390.88,A -85,B 0,C 180,E1 -1175.939,E2 -1175.939} C_VEL
LIN {X 0,Y 594.307,Z 384.24,A -85,B 0,C 180,E1 -1176.962,E2 -1176.962} C_VEL
LIN {X 0,Y 594.359,Z 375.994,A -85,B 0,C 180,E1 -1177.986,E2 -1177.986} C_VEL
LIN {X 0,Y 594.382,Z 367.543,A -85,B 0,C 180,E1 -1178.842,E2 -1178.842} C_VEL
LIN {X 0,Y 594.433,Z 357.102,A -85,B 0,C 180,E1 -1179.699,E2 -1179.699} C_VEL
LIN {X 0,Y 594.492,Z 346.767,A -85,B 0,C 180,E1 -1180.386,E2 -1180.386} C_VEL
LIN {X 0,Y 594.562,Z 335.681,A -85,B 0,C 180,E1 -1180.975,E2 -1180.975} C_VEL
LIN {X 0,Y 594.6,Z 323.712,A -85,B 0,C 180,E1 -1181.464,E2 -1181.464} C_VEL
LIN {X 0,Y 594.654,Z 310.375,A -85,B 0,C 180,E1 -1181.849,E2 -1181.849} C_VEL
LIN {X 0,Y 594.695,Z 297.128,A -85,B 0,C 180,E1 -1182.086,E2 -1182.086} C_VEL
LIN {X 0,Y 594.63,Z 196.982,A -85,B 0,C 180,E1 -1183.303,E2 -1183.303} C_VEL
LIN {X 0,Y 594.424,Z 195.103,A -85,B 0,C 180,E1 -1183.372,E2 -1183.372} C_VEL
LIN {X 0,Y 594.481,Z 176.296,A -85,B 0,C 180,E1 -1186.129,E2 -1186.129} C_VEL
LIN {X 0,Y 594.586,Z 157.912,A -85,B 0,C 180,E1 -1188.871,E2 -1188.871} C_VEL
LIN {X 0,Y 594.677,Z 141.634,A -85,B 0,C 180,E1 -1191.336,E2 -1191.336} C_VEL
LIN {X 0,Y 594.369,Z 139.519,A -85,B 0,C 180,E1 -1191.73,E2 -1191.73} C_VEL
LIN {X 0,Y 594.342,Z 139.445,A -85,B 0,C 180,E1 -1194.447,E2 -1194.447} C_VEL
LIN {X 0,Y 594.363,Z 139.444,A -85,B 0,C 180,E1 -1196.7,E2 -1196.7} C_VEL
LIN {X 0,Y 594.369,Z 139.447,A -85,B 0,C 180,E1 -1198.998,E2 -1198.998} C_VEL
LIN {X 0,Y 594.375,Z 139.445,A -85,B 0,C 180,E1 -1201.642,E2 -1201.642} C_VEL
LIN {X 0,Y 594.365,Z 139.443,A -85,B 0,C 180,E1 -1204.58,E2 -1204.58} C_VEL
LIN {X 0,Y 594.38,Z 139.443,A -85,B 0,C 180,E1 -1207.607,E2 -1207.607} C_VEL
LIN {X 0,Y 594.354,Z 139.445,A -85,B 0,C 180,E1 -1210.567,E2 -1210.567} C_VEL
LIN {X 0,Y 594.353,Z 139.451,A -85,B 0,C 180,E1 -1213.299,E2 -1213.299} C_VEL
LIN {X 0,Y 594.342,Z 139.445,A -85,B 0,C 180,E1 -1216.161,E2 -1216.161} C_VEL
LIN {X 0,Y 594.364,Z 139.445,A -85,B 0,C 180,E1 -1218.535,E2 -1218.535} C_VEL
LIN {X 0,Y 594.372,Z 139.446,A -85,B 0,C 180,E1 -1221.295,E2 -1221.295} C_VEL
LIN {X 0,Y 594.34,Z 139.444,A -85,B 0,C 180,E1 -1223.755,E2 -1223.755} C_VEL
LIN {X 0,Y 594.354,Z 139.444,A -85,B 0,C 180,E1 -1226.237,E2 -1226.237} C_VEL
LIN {X 0,Y 594.356,Z 139.449,A -85,B 0,C 180,E1 -1228.649,E2 -1228.649} C_VEL
LIN {X 0,Y 594.372,Z 139.449,A -85,B 0,C 180,E1 -1231.041,E2 -1231.041} C_VEL
LIN {X 0,Y 594.375,Z 139.444,A -85,B 0,C 180,E1 -1233.3,E2 -1233.3} C_VEL
LIN {X 0,Y 594.368,Z 139.444,A -85,B 0,C 180,E1 -1236.295,E2 -1236.295} C_VEL
LIN {X 0,Y 594.394,Z 139.442,A -85,B 0,C 180,E1 -1239.224,E2 -1239.224} C_VEL
LIN {X 0,Y 594.333,Z 139.447,A -85,B 0,C 180,E1 -1242.094,E2 -1242.094} C_VEL
LIN {X 0,Y 594.35,Z 139.447,A -85,B 0,C 180,E1 -1244.219,E2 -1244.219} C_VEL
LIN {X 0,Y 594.355,Z 139.448,A -85,B 0,C 180,E1 -1247.017,E2 -1247.017} C_VEL
LIN {X 0,Y 594.392,Z 139.442,A -85,B 0,C 180,E1 -1249.095,E2 -1249.095} C_VEL
LIN {X 0,Y 594.361,Z 139.443,A -85,B 0,C 180,E1 -1251.843,E2 -1251.843} C_VEL
LIN {X 0,Y 594.388,Z 139.449,A -85,B 0,C 180,E1 -1254.572,E2 -1254.572} C_VEL
LIN {X 0,Y 594.39,Z 139.44,A -85,B 0,C 180,E1 -1257.289,E2 -1257.289} C_VEL
LIN {X 0,Y 594.386,Z 139.442,A -85,B 0,C 180,E1 -1260,E2 -1260} C_VEL
LIN {X 0,Y 594.409,Z 139.443,A -85,B 0,C 180,E1 -1262.711,E2 -1262.711} C_VEL
LIN {X 0,Y 594.372,Z 139.441,A -85,B 0,C 180,E1 -1265.428,E2 -1265.428} C_VEL
LIN {X 0,Y 594.399,Z 139.444,A -85,B 0,C 180,E1 -1268.157,E2 -1268.157} C_VEL
LIN {X 0,Y 594.386,Z 139.44,A -85,B 0,C 180,E1 -1271.08,E2 -1271.08} C_VEL
LIN {X 0,Y 594.364,Z 139.444,A -85,B 0,C 180,E1 -1273.679,E2 -1273.679} C_VEL
LIN {X 0,Y 594.346,Z 139.444,A -85,B 0,C 180,E1 -1275.347,E2 -1275.347} C_VEL
LIN {X 0,Y 593.671,Z 139.533,A -85,B 0,C 180,E1 -1275.913,E2 -1275.913} C_VEL
LIN {X 0,Y 590.803,Z 139.893,A -85,B 0,C 180,E1 -1276.831,E2 -1276.831} C_VEL
LIN {X 0,Y 588.394,Z 140.195,A -85,B 0,C 180,E1 -1277.57,E2 -1277.57} C_VEL
LIN {X 0,Y 587.374,Z 140.321,A -85,B 0,C 180,E1 -1278.14,E2 -1278.14} C_VEL
LIN {X 0,Y 587.299,Z 140.327,A -85,B 0,C 180,E1 -1278.333,E2 -1278.333} C_VEL
LIN {X 0,Y 587.346,Z 140.316,A -85,B 0,C 180,E1 -1281.045,E2 -1281.045} C_VEL
LIN {X 0,Y 587.316,Z 140.32,A -85,B 0,C 180,E1 -1283.259,E2 -1283.259} C_VEL
LIN {X 0,Y 587.313,Z 140.322,A -85,B 0,C 180,E1 -1285.518,E2 -1285.518} C_VEL
LIN {X 0,Y 587.339,Z 140.322,A -85,B 0,C 180,E1 -1287.818,E2 -1287.818} C_VEL
LIN {X 0,Y 587.335,Z 140.322,A -85,B 0,C 180,E1 -1290.512,E2 -1290.512} C_VEL
LIN {X 0,Y 587.323,Z 140.319,A -85,B 0,C 180,E1 -1293.398,E2 -1293.398} C_VEL
LIN {X 0,Y 587.309,Z 140.325,A -85,B 0,C 180,E1 -1295.899,E2 -1295.899} C_VEL
LIN {X 0,Y 587.32,Z 140.323,A -85,B 0,C 180,E1 -1298.48,E2 -1298.48} C_VEL
LIN {X 0,Y 587.326,Z 140.319,A -85,B 0,C 180,E1 -1301.158,E2 -1301.158} C_VEL
LIN {X 0,Y 587.319,Z 140.327,A -85,B 0,C 180,E1 -1304.114,E2 -1304.114} C_VEL
LIN {X 0,Y 587.304,Z 140.322,A -85,B 0,C 180,E1 -1306.994,E2 -1306.994} C_VEL
LIN {X 0,Y 587.306,Z 140.329,A -85,B 0,C 180,E1 -1309.747,E2 -1309.747} C_VEL
LIN {X 0,Y 587.339,Z 140.32,A -85,B 0,C 180,E1 -1312.393,E2 -1312.393} C_VEL
LIN {X 0,Y 587.319,Z 140.319,A -85,B 0,C 180,E1 -1314.945,E2 -1314.945} C_VEL
LIN {X 0,Y 587.333,Z 140.323,A -85,B 0,C 180,E1 -1317.422,E2 -1317.422} C_VEL
LIN {X 0,Y 587.33,Z 140.328,A -85,B 0,C 180,E1 -1319.831,E2 -1319.831} C_VEL
LIN {X 0,Y 587.34,Z 140.32,A -85,B 0,C 180,E1 -1322.31,E2 -1322.31} C_VEL
LIN {X 0,Y 587.33,Z 140.32,A -85,B 0,C 180,E1 -1324.484,E2 -1324.484} C_VEL
LIN {X 0,Y 587.337,Z 140.326,A -85,B 0,C 180,E1 -1327.487,E2 -1327.487} C_VEL
LIN {X 0,Y 587.388,Z 140.509,A -85,B 0,C 180,E1 -1329.286,E2 -1329.286} C_VEL
LIN {X 0,Y 587.621,Z 145.158,A -85,B 0,C 180,E1 -1330.071,E2 -1330.071} C_VEL
LIN {X 0,Y 587.467,Z 162.925,A -85,B 0,C 180,E1 -1332.937,E2 -1332.937} C_VEL
LIN {X 0,Y 587.391,Z 178.713,A -85,B 0,C 180,E1 -1335.449,E2 -1335.449} C_VEL
LIN {X 0,Y 587.377,Z 185.742,A -85,B 0,C 180,E1 -1336.53,E2 -1336.53} C_VEL
LIN {X 0,Y 587.775,Z 188.691,A -85,B 0,C 180,E1 -1336.605,E2 -1336.605} C_VEL
LIN {X 0,Y 587.769,Z 292.913,A -85,B 0,C 180,E1 -1337.9,E2 -1337.9} C_VEL
LIN {X 0,Y 587.694,Z 306.191,A -85,B 0,C 180,E1 -1338.205,E2 -1338.205} C_VEL
LIN {X 0,Y 587.629,Z 318.75,A -85,B 0,C 180,E1 -1338.635,E2 -1338.635} C_VEL
LIN {X 0,Y 587.565,Z 329.788,A -85,B 0,C 180,E1 -1339.142,E2 -1339.142} C_VEL
LIN {X 0,Y 587.473,Z 341.544,A -85,B 0,C 180,E1 -1339.837,E2 -1339.837} C_VEL
LIN {X 0,Y 587.392,Z 352.056,A -85,B 0,C 180,E1 -1340.618,E2 -1340.618} C_VEL
LIN {X 0,Y 587.323,Z 360.657,A -85,B 0,C 180,E1 -1341.398,E2 -1341.398} C_VEL
LIN {X 0,Y 587.274,Z 368.581,A -85,B 0,C 180,E1 -1342.263,E2 -1342.263} C_VEL
LIN {X 0,Y 587.235,Z 375.152,A -85,B 0,C 180,E1 -1343.127,E2 -1343.127} C_VEL
LIN {X 0,Y 587.237,Z 381.621,A -85,B 0,C 180,E1 -1344.162,E2 -1344.162} C_VEL
LIN {X 0,Y 587.146,Z 386.76,A -85,B 0,C 180,E1 -1345.194,E2 -1345.194} C_VEL
LIN {X 0,Y 587.212,Z 390.749,A -85,B 0,C 180,E1 -1346.226,E2 -1346.226} C_VEL
LIN {X 0,Y 587.131,Z 393.698,A -85,B 0,C 180,E1 -1347.256,E2 -1347.256} C_VEL
LIN {X 0,Y 587.141,Z 395.127,A -85,B 0,C 180,E1 -1347.942,E2 -1347.942} C_VEL
LIN {X 0,Y 587.14,Z 396.754,A -85,B 0,C 180,E1 -1349.314,E2 -1349.314} C_VEL
LIN {X 0,Y 587.137,Z 396.996,A -85,B 0,C 180,E1 -1350,E2 -1350} C_VEL
LIN {X 0,Y 587.14,Z 396.815,A -85,B 0,C 180,E1 -1350.686,E2 -1350.686} C_VEL
LIN {X 0,Y 587.141,Z 395.273,A -85,B 0,C 180,E1 -1352.058,E2 -1352.058} C_VEL
LIN {X 0,Y 587.133,Z 393.912,A -85,B 0,C 180,E1 -1352.745,E2 -1352.745} C_VEL
LIN {X 0,Y 587.213,Z 391.035,A -85,B 0,C 180,E1 -1353.774,E2 -1353.774} C_VEL
LIN {X 0,Y 587.147,Z 387.135,A -85,B 0,C 180,E1 -1354.807,E2 -1354.807} C_VEL
LIN {X 0,Y 587.23,Z 382.104,A -85,B 0,C 180,E1 -1355.839,E2 -1355.839} C_VEL
LIN {X 0,Y 587.23,Z 375.783,A -85,B 0,C 180,E1 -1356.874,E2 -1356.874} C_VEL
LIN {X 0,Y 587.288,Z 367.864,A -85,B 0,C 180,E1 -1357.91,E2 -1357.91} C_VEL
LIN {X 0,Y 587.343,Z 358.016,A -85,B 0,C 180,E1 -1358.949,E2 -1358.949} C_VEL
LIN {X 0,Y 587.421,Z 347.697,A -85,B 0,C 180,E1 -1359.816,E2 -1359.816} C_VEL
LIN {X 0,Y 587.498,Z 336.065,A -85,B 0,C 180,E1 -1360.598,E2 -1360.598} C_VEL
LIN {X 0,Y 587.585,Z 325.175,A -85,B 0,C 180,E1 -1361.177,E2 -1361.177} C_VEL
LIN {X 0,Y 587.638,Z 312.458,A -85,B 0,C 180,E1 -1361.689,E2 -1361.689} C_VEL
LIN {X 0,Y 587.711,Z 299.488,A -85,B 0,C 180,E1 -1362.058,E2 -1362.058} C_VEL
LIN {X 0,Y 587.765,Z 287.171,A -85,B 0,C 180,E1 -1362.276,E2 -1362.276} C_VEL
LIN {X 0,Y 587.665,Z 188.017,A -85,B 0,C 180,E1 -1363.495,E2 -1363.495} C_VEL
LIN {X 0,Y 587.384,Z 185.774,A -85,B 0,C 180,E1 -1363.558,E2 -1363.558} C_VEL
LIN {X 0,Y 587.448,Z 168.088,A -85,B 0,C 180,E1 -1366.328,E2 -1366.328} C_VEL
LIN {X 0,Y 587.567,Z 150.812,A -85,B 0,C 180,E1 -1369.102,E2 -1369.102} C_VEL
LIN {X 0,Y 587.516,Z 141.231,A -85,B 0,C 180,E1 -1370.664,E2 -1370.664} C_VEL
LIN {X 0,Y 587.369,Z 140.388,A -85,B 0,C 180,E1 -1370.852,E2 -1370.852} C_VEL
LIN {X 0,Y 587.315,Z 140.322,A -85,B 0,C 180,E1 -1373.259,E2 -1373.259} C_VEL
LIN {X 0,Y 587.333,Z 140.319,A -85,B 0,C 180,E1 -1375.516,E2 -1375.516} C_VEL
LIN {X 0,Y 587.341,Z 140.32,A -85,B 0,C 180,E1 -1377.818,E2 -1377.818} C_VEL
LIN {X 0,Y 587.335,Z 140.325,A -85,B 0,C 180,E1 -1380.509,E2 -1380.509} C_VEL
LIN {X 0,Y 587.334,Z 140.319,A -85,B 0,C 180,E1 -1383.396,E2 -1383.396} C_VEL
LIN {X 0,Y 587.316,Z 140.324,A -85,B 0,C 180,E1 -1385.898,E2 -1385.898} C_VEL
LIN {X 0,Y 587.32,Z 140.325,A -85,B 0,C 180,E1 -1388.479,E2 -1388.479} C_VEL
LIN {X 0,Y 587.333,Z 140.317,A -85,B 0,C 180,E1 -1391.156,E2 -1391.156} C_VEL
LIN {X 0,Y 587.325,Z 140.33,A -85,B 0,C 180,E1 -1394.113,E2 -1394.113} C_VEL
LIN {X 0,Y 587.309,Z 140.319,A -85,B 0,C 180,E1 -1396.993,E2 -1396.993} C_VEL
LIN {X 0,Y 587.317,Z 140.325,A -85,B 0,C 180,E1 -1399.746,E2 -1399.746} C_VEL
LIN {X 0,Y 587.338,Z 140.321,A -85,B 0,C 180,E1 -1402.392,E2 -1402.392} C_VEL
LIN {X 0,Y 587.32,Z 140.316,A -85,B 0,C 180,E1 -1404.944,E2 -1404.944} C_VEL
LIN {X 0,Y 587.334,Z 140.319,A -85,B 0,C 180,E1 -1407.42,E2 -1407.42} C_VEL
LIN {X 0,Y 587.327,Z 140.328,A -85,B 0,C 180,E1 -1409.829,E2 -1409.829} C_VEL
LIN {X 0,Y 587.346,Z 140.32,A -85,B 0,C 180,E1 -1412.306,E2 -1412.306} C_VEL
LIN {X 0,Y 587.34,Z 140.319,A -85,B 0,C 180,E1 -1415.241,E2 -1415.241} C_VEL
LIN {X 0,Y 587.313,Z 140.324,A -85,B 0,C 180,E1 -1418.225,E2 -1418.225} C_VEL
LIN {X 0,Y 587.344,Z 140.318,A -85,B 0,C 180,E1 -1421.151,E2 -1421.151} C_VEL
LIN {X 0,Y 587.314,Z 140.325,A -85,B 0,C 180,E1 -1424.024,E2 -1424.024} C_VEL
LIN {X 0,Y 587.348,Z 140.32,A -85,B 0,C 180,E1 -1426.154,E2 -1426.154} C_VEL
LIN {X 0,Y 587.341,Z 140.318,A -85,B 0,C 180,E1 -1428.962,E2 -1428.962} C_VEL
LIN {X 0,Y 587.358,Z 140.323,A -85,B 0,C 180,E1 -1431.745,E2 -1431.745} C_VEL
LIN {X 0,Y 587.34,Z 140.317,A -85,B 0,C 180,E1 -1434.507,E2 -1434.507} C_VEL
LIN {X 0,Y 587.374,Z 140.318,A -85,B 0,C 180,E1 -1437.257,E2 -1437.257} C_VEL
LIN {X 0,Y 587.361,Z 140.318,A -85,B 0,C 180,E1 -1440,E2 -1440} C_VEL
LIN {X 0,Y 587.36,Z 140.315,A -85,B 0,C 180,E1 -1442.743,E2 -1442.743} C_VEL
LIN {X 0,Y 587.352,Z 140.326,A -85,B 0,C 180,E1 -1445.493,E2 -1445.493} C_VEL
LIN {X 0,Y 587.315,Z 140.321,A -85,B 0,C 180,E1 -1448.256,E2 -1448.256} C_VEL
LIN {X 0,Y 587.339,Z 140.323,A -85,B 0,C 180,E1 -1451.134,E2 -1451.134} C_VEL
LIN {X 0,Y 587.347,Z 140.317,A -85,B 0,C 180,E1 -1454.257,E2 -1454.257} C_VEL
LIN {X 0,Y 587.34,Z 140.325,A -85,B 0,C 180,E1 -1457.406,E2 -1457.406} C_VEL
LIN {X 0,Y 587.316,Z 140.32,A -85,B 0,C 180,E1 -1460.305,E2 -1460.305} C_VEL
LIN {X 0,Y 587.31,Z 140.33,A -85,B 0,C 180,E1 -1463.259,E2 -1463.259} C_VEL
LIN {X 0,Y 587.317,Z 140.325,A -85,B 0,C 180,E1 -1465.518,E2 -1465.518} C_VEL
LIN {X 0,Y 587.339,Z 140.319,A -85,B 0,C 180,E1 -1467.818,E2 -1467.818} C_VEL
LIN {X 0,Y 587.315,Z 140.322,A -85,B 0,C 180,E1 -1470.508,E2 -1470.508} C_VEL
LIN {X 0,Y 587.33,Z 140.328,A -85,B 0,C 180,E1 -1473.112,E2 -1473.112} C_VEL
LIN {X 0,Y 587.29,Z 140.324,A -85,B 0,C 180,E1 -1475.538,E2 -1475.538} C_VEL
LIN {X 0,Y 587.327,Z 140.318,A -85,B 0,C 180,E1 -1477.838,E2 -1477.838} C_VEL
LIN {X 0,Y 587.304,Z 140.323,A -85,B 0,C 180,E1 -1480.255,E2 -1480.255} C_VEL
LIN {X 0,Y 587.301,Z 140.33,A -85,B 0,C 180,E1 -1483.118,E2 -1483.118} C_VEL
LIN {X 0,Y 587.309,Z 140.322,A -85,B 0,C 180,E1 -1486.049,E2 -1486.049} C_VEL
LIN {X 0,Y 587.332,Z 140.328,A -85,B 0,C 180,E1 -1488.926,E2 -1488.926} C_VEL
LIN {X 0,Y 587.316,Z 140.32,A -85,B 0,C 180,E1 -1491.52,E2 -1491.52} C_VEL
LIN {X 0,Y 587.285,Z 140.326,A -85,B 0,C 180,E1 -1494.1,E2 -1494.1} C_VEL
LIN {X 0,Y 587.335,Z 140.327,A -85,B 0,C 180,E1 -1496.889,E2 -1496.889} C_VEL
LIN {X 0,Y 587.318,Z 140.321,A -85,B 0,C 180,E1 -1499.494,E2 -1499.494} C_VEL
LIN {X 0,Y 587.34,Z 140.321,A -85,B 0,C 180,E1 -1502.31,E2 -1502.31} C_VEL
LIN {X 0,Y 587.304,Z 140.324,A -85,B 0,C 180,E1 -1505.24,E2 -1505.24} C_VEL
LIN {X 0,Y 587.347,Z 140.473,A -85,B 0,C 180,E1 -1508.181,E2 -1508.181} C_VEL
LIN {X 0,Y 587.712,Z 143.221,A -85,B 0,C 180,E1 -1508.644,E2 -1508.644} C_VEL
LIN {X 0,Y 587.568,Z 160.835,A -85,B 0,C 180,E1 -1511.34,E2 -1511.34} C_VEL
LIN {X 0,Y 587.475,Z 177.481,A -85,B 0,C 180,E1 -1513.851,E2 -1513.851} C_VEL
LIN {X 0,Y 587.406,Z 195.363,A -85,B 0,C 180,E1 -1516.486,E2 -1516.486} C_VEL
LIN {X 0,Y 587.867,Z 198.721,A -85,B 0,C 180,E1 -1516.563,E2 -1516.563} C_VEL
LIN {X 0,Y 587.753,Z 302.946,A -85,B 0,C 180,E1 -1517.856,E2 -1517.856} C_VEL
LIN {X 0,Y 587.685,Z 316.219,A -85,B 0,C 180,E1 -1518.161,E2 -1518.161} C_VEL
LIN {X 0,Y 587.602,Z 328.771,A -85,B 0,C 180,E1 -1518.59,E2 -1518.59} C_VEL
LIN {X 0,Y 587.54,Z 340.629,A -85,B 0,C 180,E1 -1519.141,E2 -1519.141} C_VEL
LIN {X 0,Y 587.47,Z 352.202,A -85,B 0,C 180,E1 -1519.837,E2 -1519.837} C_VEL
LIN {X 0,Y 587.394,Z 362.598,A -85,B 0,C 180,E1 -1520.618,E2 -1520.618} C_VEL
LIN {X 0,Y 587.322,Z 371.111,A -85,B 0,C 180,E1 -1521.397,E2 -1521.397} C_VEL
LIN {X 0,Y 587.274,Z 378.96,A -85,B 0,C 180,E1 -1522.263,E2 -1522.263} C_VEL
LIN {X 0,Y 587.23,Z 385.468,A -85,B 0,C 180,E1 -1523.126,E2 -1523.126} C_VEL
LIN {X 0,Y 587.236,Z 391.866,A -85,B 0,C 180,E1 -1524.161,E2 -1524.161} C_VEL
LIN {X 0,Y 587.147,Z 396.949,A -85,B 0,C 180,E1 -1525.193,E2 -1525.193} C_VEL
LIN {X 0,Y 587.213,Z 400.895,A -85,B 0,C 180,E1 -1526.226,E2 -1526.226} C_VEL
LIN {X 0,Y 587.132,Z 403.808,A -85,B 0,C 180,E1 -1527.255,E2 -1527.255} C_VEL
LIN {X 0,Y 587.141,Z 405.199,A -85,B 0,C 180,E1 -1527.942,E2 -1527.942} C_VEL
LIN {X 0,Y 587.14,Z 406.784,A -85,B 0,C 180,E1 -1529.314,E2 -1529.314} C_VEL
LIN {X 0,Y 587.137,Z 407,A -85,B 0,C 180,E1 -1530,E2 -1530} C_VEL
LIN {X 0,Y 587.147,Z 406.186,A -85,B 0,C 180,E1 -1531.371,E2 -1531.371} C_VEL
LIN {X 0,Y 587.141,Z 405.201,A -85,B 0,C 180,E1 -1532.058,E2 -1532.058} C_VEL
LIN {X 0,Y 587.132,Z 403.811,A -85,B 0,C 180,E1 -1532.744,E2 -1532.744} C_VEL
LIN {X 0,Y 587.213,Z 400.897,A -85,B 0,C 180,E1 -1533.774,E2 -1533.774} C_VEL
LIN {X 0,Y 587.147,Z 396.951,A -85,B 0,C 180,E1 -1534.806,E2 -1534.806} C_VEL
LIN {X 0,Y 587.217,Z 390.88,A -85,B 0,C 180,E1 -1536.011,E2 -1536.011} C_VEL
LIN {X 0,Y 587.244,Z 384.241,A -85,B 0,C 180,E1 -1537.046,E2 -1537.046} C_VEL
LIN {X 0,Y 587.299,Z 375.995,A -85,B 0,C 180,E1 -1538.083,E2 -1538.083} C_VEL
LIN {X 0,Y 587.343,Z 367.544,A -85,B 0,C 180,E1 -1538.948,E2 -1538.948} C_VEL
LIN {X 0,Y 587.421,Z 357.104,A -85,B 0,C 180,E1 -1539.816,E2 -1539.816} C_VEL
LIN {X 0,Y 587.513,Z 346.765,A -85,B 0,C 180,E1 -1540.51,E2 -1540.51} C_VEL
LIN {X 0,Y 587.583,Z 334.81,A -85,B 0,C 180,E1 -1541.149,E2 -1541.149} C_VEL
LIN {X 0,Y 587.636,Z 322.605,A -85,B 0,C 180,E1 -1541.639,E2 -1541.639} C_VEL
LIN {X 0,Y 587.711,Z 309.459,A -85,B 0,C 180,E1 -1542.013,E2 -1542.013} C_VEL
LIN {X 0,Y 587.764,Z 297.128,A -85,B 0,C 180,E1 -1542.231,E2 -1542.231} C_VEL
LIN {X 0,Y 587.682,Z 197.207,A -85,B 0,C 180,E1 -1543.46,E2 -1543.46} C_VEL
LIN {X 0,Y 587.377,Z 195.111,A -85,B 0,C 180,E1 -1543.536,E2 -1543.536} C_VEL
LIN {X 0,Y 587.478,Z 176.296,A -85,B 0,C 180,E1 -1546.327,E2 -1546.327} C_VEL
LIN {X 0,Y 587.599,Z 159.65,A -85,B 0,C 180,E1 -1548.84,E2 -1548.84} C_VEL
LIN {X 0,Y 587.75,Z 143,A -85,B 0,C 180,E1 -1551.389,E2 -1551.389} C_VEL
LIN {X 0,Y 587.34,Z 140.393,A -85,B 0,C 180,E1 -1551.865,E2 -1551.865} C_VEL
LIN {X 0,Y 587.302,Z 140.324,A -85,B 0,C 180,E1 -1554.76,E2 -1554.76} C_VEL
LIN {X 0,Y 587.338,Z 140.322,A -85,B 0,C 180,E1 -1557.69,E2 -1557.69} C_VEL
LIN {X 0,Y 587.318,Z 140.321,A -85,B 0,C 180,E1 -1560.506,E2 -1560.506} C_VEL
LIN {X 0,Y 587.332,Z 140.327,A -85,B 0,C 180,E1 -1563.11,E2 -1563.11} C_VEL
LIN {X 0,Y 587.282,Z 140.326,A -85,B 0,C 180,E1 -1565.899,E2 -1565.899} C_VEL
LIN {X 0,Y 587.313,Z 140.32,A -85,B 0,C 180,E1 -1568.479,E2 -1568.479} C_VEL
LIN {X 0,Y 587.329,Z 140.329,A -85,B 0,C 180,E1 -1571.156,E2 -1571.156} C_VEL
LIN {X 0,Y 587.304,Z 140.322,A -85,B 0,C 180,E1 -1574.111,E2 -1574.111} C_VEL
LIN {X 0,Y 587.3,Z 140.331,A -85,B 0,C 180,E1 -1576.992,E2 -1576.992} C_VEL
LIN {X 0,Y 587.301,Z 140.323,A -85,B 0,C 180,E1 -1579.744,E2 -1579.744} C_VEL
LIN {X 0,Y 587.332,Z 140.319,A -85,B 0,C 180,E1 -1582.391,E2 -1582.391} C_VEL
LIN {X 0,Y 587.34,Z 140.318,A -85,B 0,C 180,E1 -1585.651,E2 -1585.651} C_VEL
LIN {X 0,Y 587.327,Z 140.32,A -85,B 0,C 180,E1 -1588.23,E2 -1588.23} C_VEL
LIN {X 0,Y 587.336,Z 140.327,A -85,B 0,C 180,E1 -1590.866,E2 -1590.866} C_VEL
LIN {X 0,Y 587.323,Z 140.32,A -85,B 0,C 180,E1 -1593.721,E2 -1593.721} C_VEL
LIN {X 0,Y 587.309,Z 140.321,A -85,B 0,C 180,E1 -1595.992,E2 -1595.992} C_VEL
LIN {X 0,Y 587.305,Z 140.324,A -85,B 0,C 180,E1 -1598.225,E2 -1598.225} C_VEL
LIN {X 0,Y 587.337,Z 140.321,A -85,B 0,C 180,E1 -1601.151,E2 -1601.151} C_VEL
LIN {X 0,Y 587.306,Z 140.322,A -85,B 0,C 180,E1 -1604.024,E2 -1604.024} C_VEL
LIN {X 0,Y 587.337,Z 140.32,A -85,B 0,C 180,E1 -1606.154,E2 -1606.154} C_VEL
LIN {X 0,Y 587.399,Z 140.315,A -85,B 0,C 180,E1 -1608.964,E2 -1608.964} C_VEL
LIN {X 0,Y 587.323,Z 140.32,A -85,B 0,C 180,E1 -1611.744,E2 -1611.744} C_VEL
LIN {X 0,Y 587.35,Z 140.325,A -85,B 0,C 180,E1 -1614.507,E2 -1614.507} C_VEL
LIN {X 0,Y 587.358,Z 140.316,A -85,B 0,C 180,E1 -1617.257,E2 -1617.257} C_VEL
LIN {X 0,Y 587.356,Z 140.318,A -85,B 0,C 180,E1 -1620,E2 -1620} C_VEL
LIN {X 0,Y 587.373,Z 140.318,A -85,B 0,C 180,E1 -1622.743,E2 -1622.743} C_VEL
LIN {X 0,Y 587.337,Z 140.318,A -85,B 0,C 180,E1 -1625.493,E2 -1625.493} C_VEL
LIN {X 0,Y 587.354,Z 140.323,A -85,B 0,C 180,E1 -1628.255,E2 -1628.255} C_VEL
LIN {X 0,Y 587.349,Z 140.317,A -85,B 0,C 180,E1 -1631.142,E2 -1631.142} C_VEL
LIN {X 0,Y 587.351,Z 140.325,A -85,B 0,C 180,E1 -1634.261,E2 -1634.261} C_VEL
LIN {X 0,Y 587.335,Z 140.318,A -85,B 0,C 180,E1 -1637.407,E2 -1637.407} C_VEL
LIN {X 0,Y 587.299,Z 140.327,A -85,B 0,C 180,E1 -1638.333,E2 -1638.333} C_VEL
LIN {X 0,Y 586.659,Z 140.405,A -85,B 0,C 180,E1 -1638.905,E2 -1638.905} C_VEL
LIN {X 0,Y 583.832,Z 140.758,A -85,B 0,C 180,E1 -1639.833,E2 -1639.833} C_VEL
LIN {X 0,Y 581.42,Z 141.059,A -85,B 0,C 180,E1 -1640.581,E2 -1640.581} C_VEL
LIN {X 0,Y 580.369,Z 141.185,A -85,B 0,C 180,E1 -1641.157,E2 -1641.157} C_VEL
LIN {X 0,Y 580.276,Z 141.197,A -85,B 0,C 180,E1 -1641.352,E2 -1641.352} C_VEL
LIN {X 0,Y 580.271,Z 141.199,A -85,B 0,C 180,E1 -1643.558,E2 -1643.558} C_VEL
LIN {X 0,Y 580.274,Z 141.202,A -85,B 0,C 180,E1 -1645.85,E2 -1645.85} C_VEL
LIN {X 0,Y 580.292,Z 141.205,A -85,B 0,C 180,E1 -1648.186,E2 -1648.186} C_VEL
LIN {X 0,Y 580.28,Z 141.199,A -85,B 0,C 180,E1 -1650.697,E2 -1650.697} C_VEL
LIN {X 0,Y 580.293,Z 141.195,A -85,B 0,C 180,E1 -1653.317,E2 -1653.317} C_VEL
LIN {X 0,Y 580.266,Z 141.2,A -85,B 0,C 180,E1 -1655.761,E2 -1655.761} C_VEL
LIN {X 0,Y 580.279,Z 141.205,A -85,B 0,C 180,E1 -1658.147,E2 -1658.147} C_VEL
LIN {X 0,Y 580.291,Z 141.195,A -85,B 0,C 180,E1 -1660.844,E2 -1660.844} C_VEL
LIN {X 0,Y 580.271,Z 141.201,A -85,B 0,C 180,E1 -1663.659,E2 -1663.659} C_VEL
LIN {X 0,Y 580.266,Z 141.2,A -85,B 0,C 180,E1 -1666.611,E2 -1666.611} C_VEL
LIN {X 0,Y 580.291,Z 141.195,A -85,B 0,C 180,E1 -1669.158,E2 -1669.158} C_VEL
LIN {X 0,Y 580.284,Z 141.206,A -85,B 0,C 180,E1 -1671.928,E2 -1671.928} C_VEL
LIN {X 0,Y 580.278,Z 141.197,A -85,B 0,C 180,E1 -1674.456,E2 -1674.456} C_VEL
LIN {X 0,Y 580.287,Z 141.197,A -85,B 0,C 180,E1 -1676.976,E2 -1676.976} C_VEL
LIN {X 0,Y 580.291,Z 141.199,A -85,B 0,C 180,E1 -1679.426,E2 -1679.426} C_VEL
LIN {X 0,Y 580.289,Z 141.2,A -85,B 0,C 180,E1 -1682.144,E2 -1682.144} C_VEL
LIN {X 0,Y 580.304,Z 141.196,A -85,B 0,C 180,E1 -1684.921,E2 -1684.921} C_VEL
LIN {X 0,Y 580.27,Z 141.207,A -85,B 0,C 180,E1 -1687.948,E2 -1687.948} C_VEL
LIN {X 0,Y 580.342,Z 141.319,A -85,B 0,C 180,E1 -1689.153,E2 -1689.153} C_VEL
LIN {X 0,Y 580.67,Z 145.155,A -85,B 0,C 180,E1 -1689.823,E2 -1689.823} C_VEL
LIN {X 0,Y 580.489,Z 163.281,A -85,B 0,C 180,E1 -1692.782,E2 -1692.782} C_VEL
LIN {X 0,Y 580.368,Z 178.716,A -85,B 0,C 180,E1 -1695.269,E2 -1695.269} C_VEL
LIN {X 0,Y 580.389,Z 185.757,A -85,B 0,C 180,E1 -1696.365,E2 -1696.365} C_VEL
LIN {X 0,Y 580.882,Z 189.63,A -85,B 0,C 180,E1 -1696.455,E2 -1696.455} C_VEL
LIN {X 0,Y 580.845,Z 292.942,A -85,B 0,C 180,E1 -1697.754,E2 -1697.754} C_VEL
LIN {X 0,Y 580.744,Z 306.208,A -85,B 0,C 180,E1 -1698.062,E2 -1698.062} C_VEL
LIN {X 0,Y 580.676,Z 318.367,A -85,B 0,C 180,E1 -1698.481,E2 -1698.481} C_VEL
LIN {X 0,Y 580.605,Z 329.801,A -85,B 0,C 180,E1 -1699.01,E2 -1699.01} C_VEL
LIN {X 0,Y 580.452,Z 341.55,A -85,B 0,C 180,E1 -1699.713,E2 -1699.713} C_VEL
LIN {X 0,Y 580.344,Z 352.065,A -85,B 0,C 180,E1 -1700.503,E2 -1700.503} C_VEL
LIN {X 0,Y 580.272,Z 360.663,A -85,B 0,C 180,E1 -1701.293,E2 -1701.293} C_VEL
LIN {X 0,Y 580.222,Z 368.586,A -85,B 0,C 180,E1 -1702.169,E2 -1702.169} C_VEL
LIN {X 0,Y 580.168,Z 376.287,A -85,B 0,C 180,E1 -1703.21,E2 -1703.21} C_VEL
LIN {X 0,Y 580.139,Z 383.448,A -85,B 0,C 180,E1 -1704.439,E2 -1704.439} C_VEL
LIN {X 0,Y 580.108,Z 388.19,A -85,B 0,C 180,E1 -1705.484,E2 -1705.484} C_VEL
LIN {X 0,Y 580.123,Z 391.823,A -85,B 0,C 180,E1 -1706.528,E2 -1706.528} C_VEL
LIN {X 0,Y 580.043,Z 393.7,A -85,B 0,C 180,E1 -1707.222,E2 -1707.222} C_VEL
LIN {X 0,Y 580.04,Z 395.127,A -85,B 0,C 180,E1 -1707.917,E2 -1707.917} C_VEL
LIN {X 0,Y 580.04,Z 396.755,A -85,B 0,C 180,E1 -1709.306,E2 -1709.306} C_VEL
LIN {X 0,Y 580.038,Z 396.996,A -85,B 0,C 180,E1 -1710,E2 -1710} C_VEL
LIN {X 0,Y 580.04,Z 396.815,A -85,B 0,C 180,E1 -1710.695,E2 -1710.695} C_VEL
LIN {X 0,Y 580.04,Z 395.27,A -85,B 0,C 180,E1 -1712.083,E2 -1712.083} C_VEL
LIN {X 0,Y 580.044,Z 393.91,A -85,B 0,C 180,E1 -1712.778,E2 -1712.778} C_VEL
LIN {X 0,Y 580.11,Z 391.033,A -85,B 0,C 180,E1 -1713.821,E2 -1713.821} C_VEL
LIN {X 0,Y 580.053,Z 387.133,A -85,B 0,C 180,E1 -1714.865,E2 -1714.865} C_VEL
LIN {X 0,Y 580.162,Z 382.101,A -85,B 0,C 180,E1 -1715.91,E2 -1715.91} C_VEL
LIN {X 0,Y 580.158,Z 375.779,A -85,B 0,C 180,E1 -1716.958,E2 -1716.958} C_VEL
LIN {X 0,Y 580.241,Z 367.859,A -85,B 0,C 180,E1 -1718.007,E2 -1718.007} C_VEL
LIN {X 0,Y 580.308,Z 358.01,A -85,B 0,C 180,E1 -1719.058,E2 -1719.058} C_VEL
LIN {X 0,Y 580.421,Z 347.692,A -85,B 0,C 180,E1 -1719.936,E2 -1719.936} C_VEL
LIN {X 0,Y 580.508,Z 336.053,A -85,B 0,C 180,E1 -1720.728,E2 -1720.728} C_VEL
LIN {X 0,Y 580.626,Z 324.348,A -85,B 0,C 180,E1 -1721.35,E2 -1721.35} C_VEL
LIN {X 0,Y 580.703,Z 312.626,A -85,B 0,C 180,E1 -1721.824,E2 -1721.824} C_VEL
LIN {X 0,Y 580.783,Z 299.464,A -85,B 0,C 180,E1 -1722.204,E2 -1722.204} C_VEL
LIN {X 0,Y 580.849,Z 287.13,A -85,B 0,C 180,E1 -1722.424,E2 -1722.424} C_VEL
LIN {X 0,Y 580.766,Z 188.754,A -85,B 0,C 180,E1 -1723.649,E2 -1723.649} C_VEL
LIN {X 0,Y 580.352,Z 185.768,A -85,B 0,C 180,E1 -1723.726,E2 -1723.726} C_VEL
LIN {X 0,Y 580.453,Z 168.084,A -85,B 0,C 180,E1 -1726.531,E2 -1726.531} C_VEL
LIN {X 0,Y 580.626,Z 150.041,A -85,B 0,C 180,E1 -1729.465,E2 -1729.465} C_VEL
LIN {X 0,Y 580.65,Z 143.458,A -85,B 0,C 180,E1 -1730.549,E2 -1730.549} C_VEL
LIN {X 0,Y 580.316,Z 141.252,A -85,B 0,C 180,E1 -1730.983,E2 -1730.983} C_VEL
LIN {X 0,Y 580.274,Z 141.199,A -85,B 0,C 180,E1 -1733.558,E2 -1733.558} C_VEL
LIN {X 0,Y 580.294,Z 141.199,A -85,B 0,C 180,E1 -1735.849,E2 -1735.849} C_VEL
LIN {X 0,Y 580.296,Z 141.203,A -85,B 0,C 180,E1 -1738.185,E2 -1738.185} C_VEL
LIN {X 0,Y 580.282,Z 141.2,A -85,B 0,C 180,E1 -1740.694,E2 -1740.694} C_VEL
LIN {X 0,Y 580.304,Z 141.194,A -85,B 0,C 180,E1 -1743.316,E2 -1743.316} C_VEL
LIN {X 0,Y 580.273,Z 141.199,A -85,B 0,C 180,E1 -1745.76,E2 -1745.76} C_VEL
LIN {X 0,Y 580.284,Z 141.206,A -85,B 0,C 180,E1 -1748.146,E2 -1748.146} C_VEL
LIN {X 0,Y 580.295,Z 141.195,A -85,B 0,C 180,E1 -1750.843,E2 -1750.843} C_VEL
LIN {X 0,Y 580.276,Z 141.2,A -85,B 0,C 180,E1 -1753.657,E2 -1753.657} C_VEL
LIN {X 0,Y 580.27,Z 141.198,A -85,B 0,C 180,E1 -1756.609,E2 -1756.609} C_VEL
LIN {X 0,Y 580.296,Z 141.195,A -85,B 0,C 180,E1 -1759.156,E2 -1759.156} C_VEL
LIN {X 0,Y 580.285,Z 141.205,A -85,B 0,C 180,E1 -1761.926,E2 -1761.926} C_VEL
LIN {X 0,Y 580.279,Z 141.195,A -85,B 0,C 180,E1 -1764.454,E2 -1764.454} C_VEL
LIN {X 0,Y 580.285,Z 141.195,A -85,B 0,C 180,E1 -1766.975,E2 -1766.975} C_VEL
LIN {X 0,Y 580.289,Z 141.198,A -85,B 0,C 180,E1 -1769.425,E2 -1769.425} C_VEL
LIN {X 0,Y 580.315,Z 141.198,A -85,B 0,C 180,E1 -1772.136,E2 -1772.136} C_VEL
LIN {X 0,Y 580.313,Z 141.195,A -85,B 0,C 180,E1 -1775.27,E2 -1775.27} C_VEL
LIN {X 0,Y 580.265,Z 141.206,A -85,B 0,C 180,E1 -1777.947,E2 -1777.947} C_VEL
LIN {X 0,Y 580.293,Z 141.196,A -85,B 0,C 180,E1 -1780.913,E2 -1780.913} C_VEL
LIN {X 0,Y 580.271,Z 141.206,A -85,B 0,C 180,E1 -1783.825,E2 -1783.825} C_VEL
LIN {X 0,Y 580.315,Z 141.198,A -85,B 0,C 180,E1 -1785.983,E2 -1785.983} C_VEL
LIN {X 0,Y 580.296,Z 141.195,A -85,B 0,C 180,E1 -1788.827,E2 -1788.827} C_VEL
LIN {X 0,Y 580.323,Z 141.2,A -85,B 0,C 180,E1 -1791.644,E2 -1791.644} C_VEL
LIN {X 0,Y 580.306,Z 141.194,A -85,B 0,C 180,E1 -1794.44,E2 -1794.44} C_VEL
LIN {X 0,Y 580.338,Z 141.193,A -85,B 0,C 180,E1 -1797.223,E2 -1797.223} C_VEL
LIN {X 0,Y 580.331,Z 141.194,A -85,B 0,C 180,E1 -1800,E2 -1800} C_VEL
LIN {X 0,Y 580.328,Z 141.192,A -85,B 0,C 180,E1 -1802.777,E2 -1802.777} C_VEL
LIN {X 0,Y 580.316,Z 141.201,A -85,B 0,C 180,E1 -1805.56,E2 -1805.56} C_VEL
LIN {X 0,Y 580.313,Z 141.199,A -85,B 0,C 180,E1 -1807.656,E2 -1807.656} C_VEL
LIN {X 0,Y 580.286,Z 141.195,A -85,B 0,C 180,E1 -1810.467,E2 -1810.467} C_VEL
LIN {X 0,Y 580.291,Z 141.195,A -85,B 0,C 180,E1 -1812.592,E2 -1812.592} C_VEL
LIN {X 0,Y 580.277,Z 141.199,A -85,B 0,C 180,E1 -1814.735,E2 -1814.735} C_VEL
LIN {X 0,Y 580.282,Z 141.2,A -85,B 0,C 180,E1 -1817.625,E2 -1817.625} C_VEL
LIN {X 0,Y 580.277,Z 141.199,A -85,B 0,C 180,E1 -1819.823,E2 -1819.823} C_VEL
LIN {X 0,Y 580.259,Z 141.2,A -85,B 0,C 180,E1 -1822.053,E2 -1822.053} C_VEL
LIN {X 0,Y 580.295,Z 141.202,A -85,B 0,C 180,E1 -1825.08,E2 -1825.08} C_VEL
LIN {X 0,Y 580.291,Z 141.195,A -85,B 0,C 180,E1 -1828.186,E2 -1828.186} C_VEL
LIN {X 0,Y 580.266,Z 141.202,A -85,B 0,C 180,E1 -1830.693,E2 -1830.693} C_VEL
LIN {X 0,Y 580.277,Z 141.203,A -85,B 0,C 180,E1 -1833.314,E2 -1833.314} C_VEL
LIN {X 0,Y 580.238,Z 141.2,A -85,B 0,C 180,E1 -1835.757,E2 -1835.757} C_VEL
LIN {X 0,Y 580.278,Z 141.196,A -85,B 0,C 180,E1 -1838.147,E2 -1838.147} C_VEL
LIN {X 0,Y 580.291,Z 141.204,A -85,B 0,C 180,E1 -1840.844,E2 -1840.844} C_VEL
LIN {X 0,Y 580.237,Z 141.203,A -85,B 0,C 180,E1 -1843.662,E2 -1843.662} C_VEL
LIN {X 0,Y 580.263,Z 141.204,A -85,B 0,C 180,E1 -1846.611,E2 -1846.611} C_VEL
LIN {X 0,Y 580.287,Z 141.196,A -85,B 0,C 180,E1 -1849.73,E2 -1849.73} C_VEL
LIN {X 0,Y 580.285,Z 141.203,A -85,B 0,C 180,E1 -1852.731,E2 -1852.731} C_VEL
LIN {X 0,Y 580.288,Z 141.196,A -85,B 0,C 180,E1 -1855.443,E2 -1855.443} C_VEL
LIN {X 0,Y 580.297,Z 141.196,A -85,B 0,C 180,E1 -1857.97,E2 -1857.97} C_VEL
LIN {X 0,Y 580.282,Z 141.202,A -85,B 0,C 180,E1 -1861.024,E2 -1861.024} C_VEL
LIN {X 0,Y 580.267,Z 141.199,A -85,B 0,C 180,E1 -1863.672,E2 -1863.672} C_VEL
LIN {X 0,Y 580.255,Z 141.205,A -85,B 0,C 180,E1 -1866.441,E2 -1866.441} C_VEL
LIN {X 0,Y 580.319,Z 141.402,A -85,B 0,C 180,E1 -1868.066,E2 -1868.066} C_VEL
LIN {X 0,Y 580.779,Z 145.335,A -85,B 0,C 180,E1 -1868.714,E2 -1868.714} C_VEL
LIN {X 0,Y 580.612,Z 163.213,A -85,B 0,C 180,E1 -1871.474,E2 -1871.474} C_VEL
LIN {X 0,Y 580.451,Z 181.048,A -85,B 0,C 180,E1 -1874.191,E2 -1874.191} C_VEL
LIN {X 0,Y 580.385,Z 195.376,A -85,B 0,C 180,E1 -1876.32,E2 -1876.32} C_VEL
LIN {X 0,Y 580.979,Z 200.51,A -85,B 0,C 180,E1 -1876.423,E2 -1876.423} C_VEL
LIN {X 0,Y 580.837,Z 302.946,A -85,B 0,C 180,E1 -1877.709,E2 -1877.709} C_VEL
LIN {X 0,Y 580.756,Z 316.218,A -85,B 0,C 180,E1 -1878.017,E2 -1878.017} C_VEL
LIN {X 0,Y 580.641,Z 329.494,A -85,B 0,C 180,E1 -1878.48,E2 -1878.48} C_VEL
LIN {X 0,Y 580.563,Z 340.627,A -85,B 0,C 180,E1 -1879.009,E2 -1879.009} C_VEL
LIN {X 0,Y 580.448,Z 352.2,A -85,B 0,C 180,E1 -1879.712,E2 -1879.712} C_VEL
LIN {X 0,Y 580.345,Z 362.6,A -85,B 0,C 180,E1 -1880.503,E2 -1880.503} C_VEL
LIN {X 0,Y 580.271,Z 371.112,A -85,B 0,C 180,E1 -1881.292,E2 -1881.292} C_VEL
LIN {X 0,Y 580.222,Z 378.96,A -85,B 0,C 180,E1 -1882.168,E2 -1882.168} C_VEL
LIN {X 0,Y 580.154,Z 386.65,A -85,B 0,C 180,E1 -1883.222,E2 -1883.222} C_VEL
LIN {X 0,Y 580.139,Z 393.679,A -85,B 0,C 180,E1 -1884.438,E2 -1884.438} C_VEL
LIN {X 0,Y 580.108,Z 398.371,A -85,B 0,C 180,E1 -1885.483,E2 -1885.483} C_VEL
LIN {X 0,Y 580.123,Z 401.957,A -85,B 0,C 180,E1 -1886.527,E2 -1886.527} C_VEL
LIN {X 0,Y 580.043,Z 403.808,A -85,B 0,C 180,E1 -1887.222,E2 -1887.222} C_VEL
LIN {X 0,Y 580.04,Z 405.198,A -85,B 0,C 180,E1 -1887.917,E2 -1887.917} C_VEL
LIN {X 0,Y 580.04,Z 406.785,A -85,B 0,C 180,E1 -1889.305,E2 -1889.305} C_VEL
LIN {X 0,Y 580.037,Z 407,A -85,B 0,C 180,E1 -1890,E2 -1890} C_VEL
LIN {X 0,Y 580.046,Z 406.187,A -85,B 0,C 180,E1 -1891.388,E2 -1891.388} C_VEL
LIN {X 0,Y 580.04,Z 405.2,A -85,B 0,C 180,E1 -1892.083,E2 -1892.083} C_VEL
LIN {X 0,Y 580.043,Z 403.811,A -85,B 0,C 180,E1 -1892.778,E2 -1892.778} C_VEL
LIN {X 0,Y 580.11,Z 400.897,A -85,B 0,C 180,E1 -1893.82,E2 -1893.82} C_VEL
LIN {X 0,Y 580.053,Z 396.951,A -85,B 0,C 180,E1 -1894.865,E2 -1894.865} C_VEL
LIN {X 0,Y 580.139,Z 390.879,A -85,B 0,C 180,E1 -1896.084,E2 -1896.084} C_VEL
LIN {X 0,Y 580.184,Z 384.241,A -85,B 0,C 180,E1 -1897.132,E2 -1897.132} C_VEL
LIN {X 0,Y 580.25,Z 375.995,A -85,B 0,C 180,E1 -1898.181,E2 -1898.181} C_VEL
LIN {X 0,Y 580.308,Z 367.544,A -85,B 0,C 180,E1 -1899.058,E2 -1899.058} C_VEL
LIN {X 0,Y 580.425,Z 357.105,A -85,B 0,C 180,E1 -1899.935,E2 -1899.935} C_VEL
LIN {X 0,Y 580.516,Z 346.763,A -85,B 0,C 180,E1 -1900.639,E2 -1900.639} C_VEL
LIN {X 0,Y 580.597,Z 335.24,A -85,B 0,C 180,E1 -1901.264,E2 -1901.264} C_VEL
LIN {X 0,Y 580.68,Z 322.489,A -85,B 0,C 180,E1 -1901.784,E2 -1901.784} C_VEL
LIN {X 0,Y 580.785,Z 309.458,A -85,B 0,C 180,E1 -1902.159,E2 -1902.159} C_VEL
LIN {X 0,Y 580.84,Z 297.128,A -85,B 0,C 180,E1 -1902.379,E2 -1902.379} C_VEL
LIN {X 0,Y 580.888,Z 198.771,A -85,B 0,C 180,E1 -1903.601,E2 -1903.601} C_VEL
LIN {X 0,Y 580.386,Z 195.394,A -85,B 0,C 180,E1 -1903.68,E2 -1903.68} C_VEL
LIN {X 0,Y 580.489,Z 177.485,A -85,B 0,C 180,E1 -1906.348,E2 -1906.348} C_VEL
LIN {X 0,Y 580.641,Z 160.839,A -85,B 0,C 180,E1 -1908.891,E2 -1908.891} C_VEL
LIN {X 0,Y 580.775,Z 144.144,A -85,B 0,C 180,E1 -1911.472,E2 -1911.472} C_VEL
LIN {X 0,Y 580.315,Z 141.305,A -85,B 0,C 180,E1 -1911.957,E2 -1911.957} C_VEL
LIN {X 0,Y 580.283,Z 141.202,A -85,B 0,C 180,E1 -1915.08,E2 -1915.08} C_VEL
LIN {X 0,Y 580.285,Z 141.196,A -85,B 0,C 180,E1 -1918.185,E2 -1918.185} C_VEL
LIN {X 0,Y 580.27,Z 141.2,A -85,B 0,C 180,E1 -1920.692,E2 -1920.692} C_VEL
LIN {X 0,Y 580.297,Z 141.203,A -85,B 0,C 180,E1 -1923.315,E2 -1923.315} C_VEL
LIN {X 0,Y 580.238,Z 141.205,A -85,B 0,C 180,E1 -1925.755,E2 -1925.755} C_VEL
LIN {X 0,Y 580.277,Z 141.195,A -85,B 0,C 180,E1 -1928.146,E2 -1928.146} C_VEL
LIN {X 0,Y 580.291,Z 141.201,A -85,B 0,C 180,E1 -1930.842,E2 -1930.842} C_VEL
LIN {X 0,Y 580.263,Z 141.201,A -85,B 0,C 180,E1 -1933.658,E2 -1933.658} C_VEL
LIN {X 0,Y 580.26,Z 141.202,A -85,B 0,C 180,E1 -1936.609,E2 -1936.609} C_VEL
LIN {X 0,Y 580.288,Z 141.204,A -85,B 0,C 180,E1 -1939.155,E2 -1939.155} C_VEL
LIN {X 0,Y 580.278,Z 141.195,A -85,B 0,C 180,E1 -1941.926,E2 -1941.926} C_VEL
LIN {X 0,Y 580.244,Z 141.201,A -85,B 0,C 180,E1 -1944.452,E2 -1944.452} C_VEL
LIN {X 0,Y 580.278,Z 141.207,A -85,B 0,C 180,E1 -1946.974,E2 -1946.974} C_VEL
LIN {X 0,Y 580.272,Z 141.2,A -85,B 0,C 180,E1 -1949.424,E2 -1949.424} C_VEL
LIN {X 0,Y 580.285,Z 141.197,A -85,B 0,C 180,E1 -1952.141,E2 -1952.141} C_VEL
LIN {X 0,Y 580.308,Z 141.196,A -85,B 0,C 180,E1 -1955.269,E2 -1955.269} C_VEL
LIN {X 0,Y 580.257,Z 141.2,A -85,B 0,C 180,E1 -1957.947,E2 -1957.947} C_VEL
LIN {X 0,Y 580.306,Z 141.2,A -85,B 0,C 180,E1 -1960.914,E2 -1960.914} C_VEL
LIN {X 0,Y 580.261,Z 141.199,A -85,B 0,C 180,E1 -1963.825,E2 -1963.825} C_VEL
LIN {X 0,Y 580.304,Z 141.195,A -85,B 0,C 180,E1 -1965.982,E2 -1965.982} C_VEL
LIN {X 0,Y 580.338,Z 141.196,A -85,B 0,C 180,E1 -1968.828,E2 -1968.828} C_VEL
LIN {X 0,Y 580.294,Z 141.195,A -85,B 0,C 180,E1 -1971.643,E2 -1971.643} C_VEL
LIN {X 0,Y 580.313,Z 141.2,A -85,B 0,C 180,E1 -1974.44,E2 -1974.44} C_VEL
LIN {X 0,Y 580.325,Z 141.192,A -85,B 0,C 180,E1 -1977.223,E2 -1977.223} C_VEL
LIN {X 0,Y 580.327,Z 141.194,A -85,B 0,C 180,E1 -1980,E2 -1980} C_VEL
LIN {X 0,Y 580.337,Z 141.194,A -85,B 0,C 180,E1 -1982.777,E2 -1982.777} C_VEL
LIN {X 0,Y 580.303,Z 141.194,A -85,B 0,C 180,E1 -1985.56,E2 -1985.56} C_VEL
LIN {X 0,Y 580.319,Z 141.201,A -85,B 0,C 180,E1 -1988.356,E2 -1988.356} C_VEL
LIN {X 0,Y 580.32,Z 141.192,A -85,B 0,C 180,E1 -1991.209,E2 -1991.209} C_VEL
LIN {X 0,Y 580.301,Z 141.203,A -85,B 0,C 180,E1 -1994.339,E2 -1994.339} C_VEL
LIN {X 0,Y 580.302,Z 141.195,A -85,B 0,C 180,E1 -1996.916,E2 -1996.916} C_VEL
LIN {X 0,Y 580.294,Z 141.199,A -85,B 0,C 180,E1 -1999.823,E2 -1999.823} C_VEL
LIN {X 0,Y 580.276,Z 141.197,A -85,B 0,C 180,E1 -2001.352,E2 -2001.352} C_VEL
LIN {X 0,Y 579.582,Z 141.29,A -85,B 0,C 180,E1 -2001.932,E2 -2001.932} C_VEL
LIN {X 0,Y 576.705,Z 141.644,A -85,B 0,C 180,E1 -2002.871,E2 -2002.871} C_VEL
LIN {X 0,Y 574.307,Z 141.942,A -85,B 0,C 180,E1 -2003.628,E2 -2003.628} C_VEL
LIN {X 0,Y 573.306,Z 142.076,A -85,B 0,C 180,E1 -2004.212,E2 -2004.212} C_VEL
LIN {X 0,Y 573.239,Z 142.076,A -85,B 0,C 180,E1 -2004.409,E2 -2004.409} C_VEL
LIN {X 0,Y 573.238,Z 142.074,A -85,B 0,C 180,E1 -2006.977,E2 -2006.977} C_VEL
LIN {X 0,Y 573.241,Z 142.075,A -85,B 0,C 180,E1 -2009.49,E2 -2009.49} C_VEL
LIN {X 0,Y 573.244,Z 142.074,A -85,B 0,C 180,E1 -2012.646,E2 -2012.646} C_VEL
LIN {X 0,Y 573.244,Z 142.068,A -85,B 0,C 180,E1 -2015.186,E2 -2015.186} C_VEL
LIN {X 0,Y 573.227,Z 142.08,A -85,B 0,C 180,E1 -2017.808,E2 -2017.808} C_VEL
LIN {X 0,Y 573.262,Z 142.073,A -85,B 0,C 180,E1 -2020.529,E2 -2020.529} C_VEL
LIN {X 0,Y 573.237,Z 142.077,A -85,B 0,C 180,E1 -2023.67,E2 -2023.67} C_VEL
LIN {X 0,Y 573.229,Z 142.076,A -85,B 0,C 180,E1 -2026.642,E2 -2026.642} C_VEL
LIN {X 0,Y 573.239,Z 142.077,A -85,B 0,C 180,E1 -2029.476,E2 -2029.476} C_VEL
LIN {X 0,Y 573.23,Z 142.08,A -85,B 0,C 180,E1 -2032.193,E2 -2032.193} C_VEL
LIN {X 0,Y 573.247,Z 142.072,A -85,B 0,C 180,E1 -2034.816,E2 -2034.816} C_VEL
LIN {X 0,Y 573.25,Z 142.077,A -85,B 0,C 180,E1 -2037.356,E2 -2037.356} C_VEL
LIN {X 0,Y 573.242,Z 142.075,A -85,B 0,C 180,E1 -2040.513,E2 -2040.513} C_VEL
LIN {X 0,Y 573.216,Z 142.079,A -85,B 0,C 180,E1 -2043.023,E2 -2043.023} C_VEL
LIN {X 0,Y 573.273,Z 142.076,A -85,B 0,C 180,E1 -2045.367,E2 -2045.367} C_VEL
LIN {X 0,Y 573.228,Z 142.08,A -85,B 0,C 180,E1 -2048.42,E2 -2048.42} C_VEL
LIN {X 0,Y 573.303,Z 142.223,A -85,B 0,C 180,E1 -2049.046,E2 -2049.046} C_VEL
LIN {X 0,Y 573.699,Z 146.253,A -85,B 0,C 180,E1 -2049.754,E2 -2049.754} C_VEL
LIN {X 0,Y 573.482,Z 164.179,A -85,B 0,C 180,E1 -2052.712,E2 -2052.712} C_VEL
LIN {X 0,Y 573.363,Z 180.749,A -85,B 0,C 180,E1 -2055.414,E2 -2055.414} C_VEL
LIN {X 0,Y 573.364,Z 185.775,A -85,B 0,C 180,E1 -2056.194,E2 -2056.194} C_VEL
LIN {X 0,Y 574.013,Z 190.57,A -85,B 0,C 180,E1 -2056.301,E2 -2056.301} C_VEL
LIN {X 0,Y 573.91,Z 292.971,A -85,B 0,C 180,E1 -2057.604,E2 -2057.604} C_VEL
LIN {X 0,Y 573.82,Z 306.226,A -85,B 0,C 180,E1 -2057.916,E2 -2057.916} C_VEL
LIN {X 0,Y 573.716,Z 318.382,A -85,B 0,C 180,E1 -2058.34,E2 -2058.34} C_VEL
LIN {X 0,Y 573.622,Z 329.869,A -85,B 0,C 180,E1 -2058.877,E2 -2058.877} C_VEL
LIN {X 0,Y 573.438,Z 341.556,A -85,B 0,C 180,E1 -2059.586,E2 -2059.586} C_VEL
LIN {X 0,Y 573.331,Z 352.073,A -85,B 0,C 180,E1 -2060.386,E2 -2060.386} C_VEL
LIN {X 0,Y 573.241,Z 360.669,A -85,B 0,C 180,E1 -2061.185,E2 -2061.185} C_VEL
LIN {X 0,Y 573.161,Z 368.59,A -85,B 0,C 180,E1 -2062.072,E2 -2062.072} C_VEL
LIN {X 0,Y 573.092,Z 376.526,A -85,B 0,C 180,E1 -2063.163,E2 -2063.163} C_VEL
LIN {X 0,Y 573.07,Z 383.451,A -85,B 0,C 180,E1 -2064.37,E2 -2064.37} C_VEL
LIN {X 0,Y 573.028,Z 388.192,A -85,B 0,C 180,E1 -2065.428,E2 -2065.428} C_VEL
LIN {X 0,Y 573.022,Z 391.825,A -85,B 0,C 180,E1 -2066.485,E2 -2066.485} C_VEL
LIN {X 0,Y 572.959,Z 393.702,A -85,B 0,C 180,E1 -2067.188,E2 -2067.188} C_VEL
LIN {X 0,Y 572.939,Z 395.127,A -85,B 0,C 180,E1 -2067.891,E2 -2067.891} C_VEL
LIN {X 0,Y 572.941,Z 396.756,A -85,B 0,C 180,E1 -2069.297,E2 -2069.297} C_VEL
LIN {X 0,Y 572.939,Z 396.996,A -85,B 0,C 180,E1 -2070,E2 -2070} C_VEL
LIN {X 0,Y 572.94,Z 396.815,A -85,B 0,C 180,E1 -2070.703,E2 -2070.703} C_VEL
LIN {X 0,Y 572.94,Z 395.268,A -85,B 0,C 180,E1 -2072.109,E2 -2072.109} C_VEL
LIN {X 0,Y 572.96,Z 393.908,A -85,B 0,C 180,E1 -2072.813,E2 -2072.813} C_VEL
LIN {X 0,Y 573.015,Z 391.031,A -85,B 0,C 180,E1 -2073.868,E2 -2073.868} C_VEL
LIN {X 0,Y 572.963,Z 387.131,A -85,B 0,C 180,E1 -2074.926,E2 -2074.926} C_VEL
LIN {X 0,Y 573.076,Z 382.099,A -85,B 0,C 180,E1 -2075.984,E2 -2075.984} C_VEL
LIN {X 0,Y 573.083,Z 375.775,A -85,B 0,C 180,E1 -2077.044,E2 -2077.044} C_VEL
LIN {X 0,Y 573.175,Z 367.854,A -85,B 0,C 180,E1 -2078.106,E2 -2078.106} C_VEL
LIN {X 0,Y 573.287,Z 358.003,A -85,B 0,C 180,E1 -2079.17,E2 -2079.17} C_VEL
LIN {X 0,Y 573.423,Z 347.687,A -85,B 0,C 180,E1 -2080.058,E2 -2080.058} C_VEL
LIN {X 0,Y 573.508,Z 336.077,A -85,B 0,C 180,E1 -2080.858,E2 -2080.858} C_VEL
LIN {X 0,Y 573.658,Z 325.198,A -85,B 0,C 180,E1 -2081.449,E2 -2081.449} C_VEL
LIN {X 0,Y 573.746,Z 312.61,A -85,B 0,C 180,E1 -2081.97,E2 -2081.97} C_VEL
LIN {X 0,Y 573.845,Z 299.44,A -85,B 0,C 180,E1 -2082.354,E2 -2082.354} C_VEL
LIN {X 0,Y 573.926,Z 287.089,A -85,B 0,C 180,E1 -2082.576,E2 -2082.576} C_VEL
LIN {X 0,Y 573.873,Z 189.491,A -85,B 0,C 180,E1 -2083.806,E2 -2083.806} C_VEL
LIN {X 0,Y 573.342,Z 185.763,A -85,B 0,C 180,E1 -2083.897,E2 -2083.897} C_VEL
LIN {X 0,Y 573.448,Z 168.215,A -85,B 0,C 180,E1 -2086.717,E2 -2086.717} C_VEL
LIN {X 0,Y 573.641,Z 150.384,A -85,B 0,C 180,E1 -2089.652,E2 -2089.652} C_VEL
LIN {X 0,Y 573.672,Z 144.552,A -85,B 0,C 180,E1 -2090.623,E2 -2090.623} C_VEL
LIN {X 0,Y 573.282,Z 142.123,A -85,B 0,C 180,E1 -2091.086,E2 -2091.086} C_VEL
LIN {X 0,Y 573.229,Z 142.079,A -85,B 0,C 180,E1 -2093.865,E2 -2093.865} C_VEL
LIN {X 0,Y 573.239,Z 142.083,A -85,B 0,C 180,E1 -2096.492,E2 -2096.492} C_VEL
LIN {X 0,Y 573.262,Z 142.072,A -85,B 0,C 180,E1 -2099.366,E2 -2099.366} C_VEL
LIN {X 0,Y 573.251,Z 142.08,A -85,B 0,C 180,E1 -2102.228,E2 -2102.228} C_VEL
LIN {X 0,Y 573.237,Z 142.075,A -85,B 0,C 180,E1 -2104.771,E2 -2104.771} C_VEL
LIN {X 0,Y 573.251,Z 142.073,A -85,B 0,C 180,E1 -2107.165,E2 -2107.165} C_VEL
LIN {X 0,Y 573.236,Z 142.075,A -85,B 0,C 180,E1 -2109.607,E2 -2109.607} C_VEL
LIN {X 0,Y 573.237,Z 142.077,A -85,B 0,C 180,E1 -2112.641,E2 -2112.641} C_VEL
LIN {X 0,Y 573.225,Z 142.078,A -85,B 0,C 180,E1 -2115.665,E2 -2115.665} C_VEL
LIN {X 0,Y 573.23,Z 142.078,A -85,B 0,C 180,E1 -2118.543,E2 -2118.543} C_VEL
LIN {X 0,Y 573.236,Z 142.075,A -85,B 0,C 180,E1 -2121.298,E2 -2121.298} C_VEL
LIN {X 0,Y 573.24,Z 142.079,A -85,B 0,C 180,E1 -2124.013,E2 -2124.013} C_VEL
LIN {X 0,Y 573.264,Z 142.071,A -85,B 0,C 180,E1 -2126.517,E2 -2126.517} C_VEL
LIN {X 0,Y 573.222,Z 142.077,A -85,B 0,C 180,E1 -2129.117,E2 -2129.117} C_VEL
LIN {X 0,Y 573.259,Z 142.08,A -85,B 0,C 180,E1 -2131.968,E2 -2131.968} C_VEL
LIN {X 0,Y 573.239,Z 142.075,A -85,B 0,C 180,E1 -2134.589,E2 -2134.589} C_VEL
LIN {X 0,Y 573.228,Z 142.082,A -85,B 0,C 180,E1 -2137.662,E2 -2137.662} C_VEL
LIN {X 0,Y 573.259,Z 142.072,A -85,B 0,C 180,E1 -2140.67,E2 -2140.67} C_VEL
LIN {X 0,Y 573.249,Z 142.08,A -85,B 0,C 180,E1 -2143.622,E2 -2143.622} C_VEL
LIN {X 0,Y 573.264,Z 142.08,A -85,B 0,C 180,E1 -2145.807,E2 -2145.807} C_VEL
LIN {X 0,Y 573.254,Z 142.072,A -85,B 0,C 180,E1 -2148.745,E2 -2148.745} C_VEL
LIN {X 0,Y 573.279,Z 142.075,A -85,B 0,C 180,E1 -2151.54,E2 -2151.54} C_VEL
LIN {X 0,Y 573.274,Z 142.07,A -85,B 0,C 180,E1 -2154.372,E2 -2154.372} C_VEL
LIN {X 0,Y 573.291,Z 142.071,A -85,B 0,C 180,E1 -2157.892,E2 -2157.892} C_VEL
LIN {X 0,Y 573.32,Z 142.064,A -85,B 0,C 180,E1 -2160.702,E2 -2160.702} C_VEL
LIN {X 0,Y 573.232,Z 142.083,A -85,B 0,C 180,E1 -2163.515,E2 -2163.515} C_VEL
LIN {X 0,Y 573.281,Z 142.076,A -85,B 0,C 180,E1 -2165.628,E2 -2165.628} C_VEL
LIN {X 0,Y 573.26,Z 142.076,A -85,B 0,C 180,E1 -2167.75,E2 -2167.75} C_VEL
LIN {X 0,Y 573.254,Z 142.072,A -85,B 0,C 180,E1 -2170.597,E2 -2170.597} C_VEL
LIN {X 0,Y 573.252,Z 142.073,A -85,B 0,C 180,E1 -2172.749,E2 -2172.749} C_VEL
LIN {X 0,Y 573.225,Z 142.08,A -85,B 0,C 180,E1 -2174.92,E2 -2174.92} C_VEL
LIN {X 0,Y 573.232,Z 142.075,A -85,B 0,C 180,E1 -2177.849,E2 -2177.849} C_VEL
LIN {X 0,Y 573.232,Z 142.075,A -85,B 0,C 180,E1 -2180.077,E2 -2180.077} C_VEL
LIN {X 0,Y 573.225,Z 142.076,A -85,B 0,C 180,E1 -2182.338,E2 -2182.338} C_VEL
LIN {X 0,Y 573.238,Z 142.081,A -85,B 0,C 180,E1 -2185.411,E2 -2185.411} C_VEL
LIN {X 0,Y 573.243,Z 142.073,A -85,B 0,C 180,E1 -2188.029,E2 -2188.029} C_VEL
LIN {X 0,Y 573.215,Z 142.083,A -85,B 0,C 180,E1 -2190.881,E2 -2190.881} C_VEL
LIN {X 0,Y 573.235,Z 142.077,A -85,B 0,C 180,E1 -2193.521,E2 -2193.521} C_VEL
LIN {X 0,Y 573.208,Z 142.074,A -85,B 0,C 180,E1 -2196.052,E2 -2196.052} C_VEL
LIN {X 0,Y 573.232,Z 142.078,A -85,B 0,C 180,E1 -2198.703,E2 -2198.703} C_VEL
LIN {X 0,Y 573.221,Z 142.078,A -85,B 0,C 180,E1 -2201.593,E2 -2201.593} C_VEL
LIN {X 0,Y 573.213,Z 142.079,A -85,B 0,C 180,E1 -2204.336,E2 -2204.336} C_VEL
LIN {X 0,Y 573.22,Z 142.08,A -85,B 0,C 180,E1 -2207.361,E2 -2207.361} C_VEL
LIN {X 0,Y 573.238,Z 142.077,A -85,B 0,C 180,E1 -2210.393,E2 -2210.393} C_VEL
LIN {X 0,Y 573.229,Z 142.082,A -85,B 0,C 180,E1 -2213.076,E2 -2213.076} C_VEL
LIN {X 0,Y 573.258,Z 142.071,A -85,B 0,C 180,E1 -2215.671,E2 -2215.671} C_VEL
LIN {X 0,Y 573.234,Z 142.077,A -85,B 0,C 180,E1 -2218.185,E2 -2218.185} C_VEL
LIN {X 0,Y 573.239,Z 142.083,A -85,B 0,C 180,E1 -2220.633,E2 -2220.633} C_VEL
LIN {X 0,Y 573.208,Z 142.082,A -85,B 0,C 180,E1 -2223.022,E2 -2223.022} C_VEL
LIN {X 0,Y 573.218,Z 142.077,A -85,B 0,C 180,E1 -2225.364,E2 -2225.364} C_VEL
LIN {X 0,Y 573.251,Z 142.246,A -85,B 0,C 180,E1 -2227.924,E2 -2227.924} C_VEL
LIN {X 0,Y 573.829,Z 146.748,A -85,B 0,C 180,E1 -2228.676,E2 -2228.676} C_VEL
LIN {X 0,Y 573.647,Z 164.381,A -85,B 0,C 180,E1 -2231.426,E2 -2231.426} C_VEL
LIN {X 0,Y 573.433,Z 182.237,A -85,B 0,C 180,E1 -2234.175,E2 -2234.175} C_VEL
LIN {X 0,Y 573.368,Z 195.388,A -85,B 0,C 180,E1 -2236.149,E2 -2236.149} C_VEL
LIN {X 0,Y 574.076,Z 200.51,A -85,B 0,C 180,E1 -2236.256,E2 -2236.256} C_VEL
LIN {X 0,Y 573.915,Z 302.946,A -85,B 0,C 180,E1 -2237.558,E2 -2237.558} C_VEL
LIN {X 0,Y 573.824,Z 315.455,A -85,B 0,C 180,E1 -2237.848,E2 -2237.848} C_VEL
LIN {X 0,Y 573.68,Z 328.376,A -85,B 0,C 180,E1 -2238.294,E2 -2238.294} C_VEL
LIN {X 0,Y 573.59,Z 340.722,A -85,B 0,C 180,E1 -2238.879,E2 -2238.879} C_VEL
LIN {X 0,Y 573.437,Z 352.197,A -85,B 0,C 180,E1 -2239.585,E2 -2239.585} C_VEL
LIN {X 0,Y 573.332,Z 362.602,A -85,B 0,C 180,E1 -2240.385,E2 -2240.385} C_VEL
LIN {X 0,Y 573.241,Z 371.112,A -85,B 0,C 180,E1 -2241.185,E2 -2241.185} C_VEL
LIN {X 0,Y 573.161,Z 378.96,A -85,B 0,C 180,E1 -2242.071,E2 -2242.071} C_VEL
LIN {X 0,Y 573.073,Z 386.954,A -85,B 0,C 180,E1 -2243.185,E2 -2243.185} C_VEL
LIN {X 0,Y 573.07,Z 393.679,A -85,B 0,C 180,E1 -2244.369,E2 -2244.369} C_VEL
LIN {X 0,Y 573.028,Z 398.372,A -85,B 0,C 180,E1 -2245.427,E2 -2245.427} C_VEL
LIN {X 0,Y 573.022,Z 401.957,A -85,B 0,C 180,E1 -2246.484,E2 -2246.484} C_VEL
LIN {X 0,Y 572.959,Z 403.807,A -85,B 0,C 180,E1 -2247.187,E2 -2247.187} C_VEL
LIN {X 0,Y 572.946,Z 406.185,A -85,B 0,C 180,E1 -2248.594,E2 -2248.594} C_VEL
LIN {X 0,Y 572.938,Z 407,A -85,B 0,C 180,E1 -2250,E2 -2250} C_VEL
